# B&R Automation Studio project Soiled_PLC (part 12)

#### ClientPanel.ab - Implementation code
```automation-basic
(********************************************************************
 * COPYRIGHT --
 ********************************************************************
 * Program: ClientPanel
 * File: ClientPanel.ab
 * Author: Dave
 * Created: December 09, 2010
 ********************************************************************
 * Implementation of program ClientPanel
 ********************************************************************)

;Version 1.00 12/12/2010 D.J. First Issue

PROGRAM _INIT

	ColdStart	= FALSE
	panelStatus = 0

	;Set IF port number for panel
	strcpy(ADR(ClientGeneral.IFport),"IF1")

END_PROGRAM

PROGRAM _CYCLIC

	;Read system information

	IF (panelStatus = 0) THEN

		IF (ClientGeneral.ChangePage <> 0) THEN
			ClientGeneral.ChangePage 	= 0 ;Set Init_Page
			ClientGeneral.ButtonPressed = 0 ;Clear button pressed
		ENDIF

		panelStatus = panelStatus + 1

	ENDIF

	;Read IP Address
	IF (panelStatus = 1) THEN

		CfgGetIPAddr_0.enable 	= TRUE
		CfgGetIPAddr_0.pDevice 	= ADR(ClientGeneral.IFport)
		CfgGetIPAddr_0.pIPAddr 	= ADR(ClientGeneral.IPaddress)
		CfgGetIPAddr_0.Len 		= SIZEOF(ClientGeneral.IPaddress)
		CfgGetIPAddr_0 FUB CfgGetIPAddr()

		IF CfgGetIPAddr_0.status = 0 THEN
			panelStatus = panelStatus + 1
		ELSE IF CfgGetIPAddr_0.status = cfgERR_DEVICE_NOT_EXIST THEN
			strcpy(ADR(ClientGeneral.IFport),"IF5") ;Try different port address IF1 = PCT03 and IF5 = CTT11
		ENDIF

	ENDIF

	;Read Subnet Mask
	IF (panelStatus = 2) THEN

		CfgGetSubnetMask_0.enable 		= TRUE
		CfgGetSubnetMask_0.pDevice 		= ADR(ClientGeneral.IFport)
		CfgGetSubnetMask_0.pSubnetMask 	= ADR(ClientGeneral.SubnetMask)
		CfgGetSubnetMask_0.Len 			= SIZEOF(ClientGeneral.SubnetMask)
		CfgGetSubnetMask_0 FUB CfgGetSubnetMask()

		IF CfgGetSubnetMask_0.status = 0 THEN
			panelStatus = panelStatus + 1
		ENDIF

	ENDIF

	;Read Gateway
	IF (panelStatus = 3) THEN

		CfgGetDefaultGateway_0.enable 	= TRUE
		CfgGetDefaultGateway_0.pDevice 	= ADR(ClientGeneral.IFport)
		CfgGetDefaultGateway_0.pGateway = ADR(ClientGeneral.Gateway)
		CfgGetDefaultGateway_0.Len 		= SIZEOF(ClientGeneral.Gateway)
		CfgGetDefaultGateway_0 FUB CfgGetDefaultGateway()

		IF CfgGetDefaultGateway_0.status = 0 THEN
			panelStatus = panelStatus + 1
		ENDIF

	ENDIF

	;Read Broadcast address
	IF (panelStatus = 4) THEN

		CfgGetBroadcastAddr_0.enable 			= TRUE
		CfgGetBroadcastAddr_0.pDevice 			= ADR(ClientGeneral.IFport)
		CfgGetBroadcastAddr_0.pBroadcastAddr 	= ADR(ClientGeneral.BroadcastAddress)
		CfgGetBroadcastAddr_0.Len 				= SIZEOF(ClientGeneral.BroadcastAddress)
		CfgGetBroadcastAddr_0 FUB CfgGetBroadcastAddr()

		IF CfgGetBroadcastAddr_0.status = 0 THEN
			panelStatus = panelStatus + 1
			ClientGeneral.ChangePage 	= 1	;Set Config Button Page
		ENDIF

	ENDIF

	;Init_Page Time Out
	TON_10ms_0.IN = (panelStatus = 5)
	TON_10ms_0.PT = 1000
	TON_10ms_0 FUB TON_10ms()

	TimedOut = TON_10ms_0.Q

	IF (panelStatus = 5) OR (panelStatus = 20) THEN
		IF (ClientGeneral.ButtonPressed = 1) THEN
			panelStatus 				= 6
			ClientGeneral.ChangePage 	= 2	;Set Password page
			ClientGeneral.ButtonPressed = 0
		ELSE IF TimedOut THEN
			panelStatus 				= 20
		ENDIF
	ENDIF

	;Password Page
	IF (panelStatus = 6)   THEN
		IF (ClientGeneral.ButtonPressed = 2) THEN
			panelStatus 				= 5
			ClientGeneral.ChangePage 	= 1	;Set Config Button Page
			ClientGeneral.ButtonPressed = 0
		ENDIF
		IF ClientGeneral.Password = 7701 THEN
			ClientGeneral.ChangePage 	= 3	;Config Page
			panelStatus 				= 7
		ENDIF
	ENDIF

	;Config Page
	IF (panelStatus = 7) THEN
		IF (ClientGeneral.ButtonPressed = 3)  THEN
			panelStatus 				= 11
			ClientGeneral.ButtonPressed = 0
		ENDIF
	ENDIF

	;Store configuration
	;-------------------

	;Store IP Address
	IF (panelStatus = 11) THEN

		CfgSetIPAddr_0.enable 	= TRUE
		CfgSetIPAddr_0.pDevice 	= ADR(ClientGeneral.IFport)
		CfgSetIPAddr_0.pIPAddr 	= ADR(ClientGeneral.IPaddress)
		CfgSetIPAddr_0.Option 	= cfgOPTION_NON_VOLATILE
		CfgSetIPAddr_0 FUB CfgSetIPAddr()

		IF CfgSetIPAddr_0.status = 0 THEN
			panelStatus = 12
		ELSE IF CfgSetIPAddr_0.status = ERR_FUB_BUSY THEN
			; Busy do Nothing
		ELSE IF CfgSetIPAddr_0.status <> ERR_FUB_BUSY THEN
			panelStatus = 12  	;Ignore Errors
		ENDIF

	ENDIF

	;Write Subnet Mask
	IF (panelStatus = 12) THEN

		CfgSetSubnetMask_0.enable 		= TRUE
		CfgSetSubnetMask_0.pDevice 		= ADR(ClientGeneral.IFport)
		CfgSetSubnetMask_0.pSubnetMask 	= ADR(ClientGeneral.SubnetMask)
		CfgSetSubnetMask_0.Option 		= cfgOPTION_NON_VOLATILE
		CfgSetSubnetMask_0 FUB CfgSetSubnetMask()

		IF CfgSetSubnetMask_0.status = 0 THEN
			panelStatus = 13
		ELSE IF CfgSetSubnetMask_0.status = ERR_FUB_BUSY THEN
			; Busy do Nothing
		ELSE IF CfgSetSubnetMask_0.status <> ERR_FUB_BUSY THEN
			panelStatus = 13 	;Ignore Errors
		ENDIF

	ENDIF

	;Write Gateway
	IF (panelStatus = 13) THEN

		CfgSetDefaultGateway_0.enable 	= TRUE
		CfgSetDefaultGateway_0.pDevice 	= ADR(ClientGeneral.IFport)
		CfgSetDefaultGateway_0.pGateway = ADR(ClientGeneral.Gateway)
		CfgSetDefaultGateway_0.Option 	= cfgOPTION_NON_VOLATILE
		CfgSetDefaultGateway_0 FUB CfgSetDefaultGateway()

		IF CfgSetDefaultGateway_0.status = 0 THEN
			panelStatus = 14
		ELSE IF CfgSetDefaultGateway_0.status = ERR_FUB_BUSY THEN
			; Busy do Nothing
		ELSE IF CfgSetDefaultGateway_0.status <> ERR_FUB_BUSY THEN
			panelStatus = 14	 ;Ignore Errors
		ENDIF

	ENDIF

	;Write Broadcast address
	IF (panelStatus = 14) THEN

		CfgSetBroadcastAddr_0.enable 			= TRUE
		CfgSetBroadcastAddr_0.pDevice 			= ADR(ClientGeneral.IFport)
		CfgSetBroadcastAddr_0.pBroadcastAddr 	= ADR(ClientGeneral.BroadcastAddress)
		CfgSetBroadcastAddr_0.Option 			= cfgOPTION_NON_VOLATILE
		CfgSetBroadcastAddr_0 FUB CfgSetBroadcastAddr()

		IF CfgSetBroadcastAddr_0.status = 0 THEN
			IF ColdStart THEN
				SysResetStatus = SYSreset(TRUE,2) ;Cold Start after changing IP address
			ELSE
				panelStatus = 20
			ENDIF
		ELSE IF CfgSetBroadcastAddr_0.status = ERR_FUB_BUSY THEN
			; Busy do Nothing
		ELSE IF CfgSetBroadcastAddr_0.status <> ERR_FUB_BUSY THEN
			IF ColdStart THEN
				SysResetStatus = SYSreset(TRUE,2) ;Cold Start after changing IP address
			ELSE
				panelStatus = 20 ;Ignore Errors
			ENDIF
		ENDIF

	ENDIF

	;Main Display Page
	IF (panelStatus = 20) THEN
		IF ClientReceive[0].MainDisplay = 0 THEN
			IF ((ClientGeneral.ChangePage <> 20) AND (ClientGeneral.CurrentPage <> 20) AND (ClientGeneral.CurrentPage <> 5)) THEN
				ClientGeneral.ChangePage = 20	;Set Default Main display page
			ENDIF
		ELSE IF ClientReceive[0].MainDisplay > 20 THEN
			IF ((ClientGeneral.ChangePage <> ClientReceive[0].MainDisplay) AND (ClientGeneral.CurrentPage <> ClientReceive[0].MainDisplay)) THEN
				ClientGeneral.ChangePage = ClientReceive[0].MainDisplay	;Set Main display page
			ENDIF
		ENDIF

		;Brightness Adjustment required?
		myBrightness = UDINT(ClientReceive[0].Brightness)
		IF (pnlBrightness <> myBrightness) THEN
			panelStatus = 21
		ENDIF

		;New IP address received
		length = strlen(ADR(ClientReceive[0].IP_Address))
		IF (length > 0) THEN
			;Copy new address before ClientReceive[0].IP_Address is cleared by the server
			strcpy(ADR(NewIPAddress),ADR(ClientReceive[0].IP_Address))
			;New IP Address is the actual Gateway
			strcpy(ADR(ClientGeneral.Gateway),ADR(ClientReceive[0].IP_Address))
			panelStatus = 31 ;Change IP Address
		ENDIF

	ENDIF

	;Remote cold Start
	IF (ClientReceive[0].SYSreset > 0) THEN
		SysResetStatus = SYSreset(TRUE,2) ;Cold Start
	ENDIF

	;Display Brightness
	IF (panelStatus = 21) THEN

		IF myVC_Handle = 0 THEN
			myVC_Handle = VA_Setup(TRUE, "Data1")
		ENDIF
		IF (myVC_Handle > 0) THEN
			IF VA_Saccess(TRUE,myVC_Handle) = 0 THEN
				VA_SetBrightness(TRUE,myVC_Handle,myBrightness)
				VA_SetBacklight(TRUE,myVC_Handle,(myBrightness > 0))
				pnlBrightness = myBrightness
				VA_Srelease(TRUE,myVC_Handle)
			ENDIF
		ENDIF

		panelStatus = 20
	ELSE
		myVC_Handle = 0
	ENDIF

	;Change IP Address
	IF (panelStatus = 31) THEN

		IP_Replace_0.pIP_New = ADR(NewIPAddress)
		IP_Replace_0.pIP_Now = ADR(ClientGeneral.IPaddress)
		IP_Replace_0 FUB IP_Replace()

		IF IP_Replace_0.status = 0 THEN
			ClientGeneral.IPaddress = IP_Replace_0.IP_Replace
			panelStatus = 32
		ELSE
			panelStatus = 20
		ENDIF

	ENDIF

	;Change Gateway
	IF (panelStatus = 32) THEN

		;IP_Replace_0.pIP_New = ADR(NewIPAddress)
		;IP_Replace_0.pIP_Now = ADR(ClientGeneral.Gateway)
		;IP_Replace_0 FUB IP_Replace()

		;IF IP_Replace_0.status = 0 THEN
		;	ClientGeneral.Gateway = IP_Replace_0.IP_Replace
			panelStatus = 33
		;ELSE
		;	panelStatus = 20
		;ENDIF

	ENDIF

	;Change Broadcast Address
	IF (panelStatus = 33) THEN

		IP_Replace_0.pIP_New = ADR(NewIPAddress)
		IP_Replace_0.pIP_Now = ADR(ClientGeneral.BroadcastAddress)
		IP_Replace_0 FUB IP_Replace()

		IF IP_Replace_0.status = 0 THEN
			ClientGeneral.BroadcastAddress = IP_Replace_0.IP_Replace
			panelStatus = 34
		ELSE
			panelStatus = 20
		ENDIF

	ENDIF

	;Change Server IP
	IF (panelStatus = 34) THEN

		IP_Replace_0.pIP_New = ADR(NewIPAddress)
		IP_Replace_0.pIP_Now = ADR(ClientServerIP)
		IP_Replace_0 FUB IP_Replace()

		IF IP_Replace_0.status = 0 THEN
			ClientServerIP 	= IP_Replace_0.IP_Replace
			ColdStart		= TRUE
			panelStatus 	= 11 ;Store New Values
		ELSE
			panelStatus = 20
		ENDIF

	ENDIF

END_PROGRAM
```

#### ClientPanel.var - Local variables
```iecst
(********************************************************************
 * COPYRIGHT --
 ********************************************************************
 * Program: ClientPanel
 * File: ClientPanel.var
 * Author: Dave
 * Created: December 09, 2010
 ********************************************************************
 * Local variables of program ClientPanel
 ********************************************************************)
VAR
	panelStatus : UINT;
	CfgGetIPAddr_0 : CfgGetIPAddr;
	CfgGetSubnetMask_0 : CfgGetSubnetMask;
	CfgGetDefaultGateway_0 : CfgGetDefaultGateway;
	CfgGetBroadcastAddr_0 : CfgGetBroadcastAddr;
	TON_10ms_0 : TON_10ms;
	TimedOut : BOOL;
	CfgSetIPAddr_0 : CfgSetIPAddr;
	CfgSetSubnetMask_0 : CfgSetSubnetMask;
	CfgSetDefaultGateway_0 : CfgSetDefaultGateway;
	CfgSetBroadcastAddr_0 : CfgSetBroadcastAddr;
	SysResetStatus : UINT;
	myVC_Handle : UDINT;
	myBrightness : UDINT;
	pnlBrightness : UDINT;
	length : UINT;
	IP_Replace_0 : IP_Replace;
	ColdStart : BOOL;
	NewIPAddress : STRING[16];
END_VAR
```

### Program Logical/Displays/Client (IEC, version 1.00.0) - AsTCP Diplay Client

#### Client.ab - Implementation code
```automation-basic
(********************************************************************
 * COPYRIGHT --
 ********************************************************************
 * Program: Client
 * File: Client.ab
 * Author: Dave
 * Created: December 06, 2010
 ********************************************************************
 * Implementation of program Client
 ********************************************************************)

;Version 1.00 12/12/2010 D.J. First Issue
;Version 2.00 22/07/2011 D.J. Added sckWaitSync - Improve Sync between Slave and Master

PROGRAM _INIT

	IF ((IdentRetain > 0) AND (Client.TcpOpen_0.ident = 0)) THEN
		Client.TcpOpen_0.ident = IdentRetain
	ENDIF

END_PROGRAM

PROGRAM _CYCLIC
	ClientText
	;Sending and Recieving Syc / Speed from Server
	ScanClock 		= clock_ms()
	ScanNow 		= (ScanClock - ScanLastClock)
	ScanLastClock 	= ScanClock
	ScanCount 		= (ScanCount + UINT(ScanNow))

	;Init Ethernet Socket - Pause after any close etc
	TON_10ms_0.IN = (SocketState = sckClosed)
	TON_10ms_0.PT = 100
	TON_10ms_0 FUB TON_10ms()

	IF TON_10ms_0.Q THEN
		SocketState = sckConnecting
	ENDIF

	;Close Ethernet Socket
	IF SocketState = sckError THEN

		Client.TcpClose_0.enable 	= TRUE
		Client.TcpClose_0.ident 	= Client.TcpOpen_0.ident
		Client.TcpClose_0.how 		= 0						;tcpSHUT_RD OR tcpSHUT_WR;
		Client.TcpClose_0 FUB TcpClose()

		IF Client.TcpClose_0.status = 0 THEN
			SocketState = sckClosed
		ELSE IF Client.TcpClose_0.status = ERR_FUB_BUSY THEN
		 	;Busy
		ELSE IF Client.TcpClose_0.status = tcpERR_INVALID_IDENT THEN
			SocketState = sckClosed
		ELSE IF Client.TcpClose_0.status = tcpERR_NOT_CONNECTED THEN
			SocketState = sckClosed
		ELSE IF Client.TcpOpen_0.status <> ERR_FUB_BUSY THEN
			SocketState = sckConnecting
		ENDIF

	ENDIF

	;Open Ethernet Socket
	IF SocketState = sckConnecting THEN
		Client.TcpOpen_0.enable  	= TRUE
		Client.TcpOpen_0.pIfAddr 	= 0					;Which Interface to open
		Client.TcpOpen_0.port 		= 12001				;Client Port
		Client.TcpOpen_0.options 	= 0
		Client.TcpOpen_0 FUB TcpOpen()

		IF Client.TcpOpen_0.status = 0 THEN
			SocketState = sckSetLinger ;sckConnected
			IdentRetain = Client.TcpOpen_0.ident
		ELSE IF Client.TcpOpen_0.status = ERR_FUB_BUSY THEN
		 	;Busy
		ELSE IF Client.TcpOpen_0.status = tcpERR_ALREADY_EXIST THEN
			SocketState = sckError
		ELSE IF Client.TcpOpen_0.status = tcpERR_SOCKET_BIND THEN
			SocketState = sckError
		ELSE
			SocketState = sckError
		ENDIF
	ENDIF

	;Set Open Linger Options
	IF SocketState = sckSetLinger THEN

		Client.linger_opt.lLinger 	= 0 ;Linger Time = 0
		Client.linger_opt.lOnOff	= 1	;Linger Option On

		Client.TcpIoctl_0.enable 	= TRUE
		Client.TcpIoctl_0.ident 	= Client.TcpOpen_0.ident
		Client.TcpIoctl_0.ioctl		= tcpSO_LINGER_SET
		Client.TcpIoctl_0.pData		= ADR(Client.linger_opt)
		Client.TcpIoctl_0.datalen 	= SIZEOF(Client.linger_opt)
		Client.TcpIoctl_0 FUB TcpIoctl()

		IF Client.TcpIoctl_0.status = 0 THEN
			SocketState = sckConnected
		ELSE IF Client.TcpIoctl_0.status = ERR_FUB_BUSY THEN  (* TcpIoctl not finished -> redo *)
			;Busy
		ELSE
			SocketState = sckError
		ENDIF
	ENDIF

	;Connect to server
	IF SocketState = sckConnected THEN

		Client.TcpClient_0.enable 	= TRUE
		Client.TcpClient_0.ident 	= Client.TcpOpen_0.ident 	;Connection Ident from AsTCP.TCP_Open
		Client.TcpClient_0.portserv = 12000						;Server port number
		Client.TcpClient_0.pServer 	= ADR(ClientServerIP)			;Server IP Adderss
		Client.TcpClient_0 FUB TcpClient()

		IF Client.TcpClient_0.status = 0 THEN
			SocketState = sckSend
		ELSE IF Client.TcpClient_0.status = ERR_FUB_BUSY THEN
			;Busy
		ELSE IF Client.TcpClient_0.status = tcpERR_INVALID THEN
			SocketState = sckError
		ELSE IF Client.TcpClient_0.status = tcpERR_NOT_CONNECTED THEN
			SocketState = sckClosed
		ELSE
			SocketState = sckError
		ENDIF

	ENDIF

	;Send Data
	IF SocketState = sckSend THEN

		Client.TcpSend_0.enable 	= TRUE
		Client.TcpSend_0.ident 		= Client.TcpOpen_0.ident
		Client.TcpSend_0.pData 		= ADR(ClientSend)	;Address of send data
		Client.TcpSend_0.datalen 	= SIZEOF(ClientSend);Length of send data
		Client.TcpSend_0.flags 		= 0
		Client.TcpSend_0 FUB TcpSend()

		IF Client.TcpSend_0.status = 0 THEN
			SocketState = sckReceive
		ELSE IF Client.TcpSend_0.status = ERR_FUB_BUSY THEN
			;Busy
		ELSE IF (Client.TcpSend_0.status = tcpERR_SENTLEN) OR (Client.TcpSend_0.status = tcpERR_NOT_CONNECTED) THEN
			SocketState = sckError
		ELSE
			SocketState = sckError
		ENDIF

	ENDIF

	IF SocketState = sckReceive THEN

		Client.TcpRecv_0.enable 	= TRUE
		Client.TcpRecv_0.ident 		= Client.TcpOpen_0.ident			;Connection Ident from AsTCP.TCP_Open
		Client.TcpRecv_0.pData		= ADR(ClientReceive)	;Where to store the incoming data
		Client.TcpRecv_0.datamax 	= SIZEOF(ClientReceive)	;Lenght of data buffer
		Client.TcpRecv_0.flags 		= 0
		Client.TcpRecv_0 FUB TcpRecv()

		IF Client.TcpRecv_0.status = 0 THEN  (* Data was received sucessfully -> Send next packet *)
			SocketState 			= sckWaitSync
		ELSE IF Client.TcpRecv_0.status = tcpERR_NO_DATA THEN  (* No data received - wait *)
		    IF Client.recv_timeout > 10 THEN
 		    	SocketState = sckError
		  	ENDIF
		ELSE IF Client.TcpRecv_0.status = ERR_FUB_BUSY THEN
			;Busy
		ELSE IF Client.TcpRecv_0.status = tcpERR_NOT_CONNECTED THEN
			SocketState = sckError
		ELSE
			SocketState = sckError
		ENDIF

		Client.recv_timeout = Client.recv_timeout + 1
	ELSE IF SocketState <> sckReceive THEN
		Client.recv_timeout = 0
	ENDIF

	;Wait until SyncStart (Master controls the connection communication speed)
	IF SocketState = sckWaitSync THEN
		IF (ScanCount >= ClientReceive[0].CycleSync_ms) THEN
			ScanCount 	= 0
			SocketState	= sckSend
		ENDIF
	ENDIF

END_PROGRAM
```

#### Client.typ - Local data types
```iecst
(********************************************************************
 * COPYRIGHT --
 ********************************************************************
 * Program: Client
 * File: Client.typ
 * Author: Dave
 * Created: December 06, 2010
 ********************************************************************
 * Local data types of program Client
 ********************************************************************)

TYPE
	Client_typ : 	STRUCT  (*TCP Client Variables*)
		TcpOpen_0 : TcpOpen; (*AsTCP.TcpOpen FUB*)
		TcpClient_0 : TcpClient; (*AsTCP.TcpClient FUB*)
		TcpRecv_0 : TcpRecv; (*AsTCP.TcpRecv FUB*)
		TcpSend_0 : TcpSend; (*AsTCP.TcpSend FUB*)
		TcpIoctl_0 : TcpIoctl; (*AsTCP.TcpIoctl FUB*)
		TcpClose_0 : TcpClose; (*AsTCP.TcpClose FUB*)
		linger_opt : tcpLINGER_typ; (*AsTCP.tcpLINGER_typ*)
		recv_timeout : UDINT; (*receive timeout*)
	END_STRUCT;
END_TYPE
```

#### Client.var - Local variables
```iecst
(********************************************************************
 * COPYRIGHT --
 ********************************************************************
 * Program: Client
 * File: Client.var
 * Author: Dave
 * Created: December 06, 2010
 ********************************************************************
 * Local variables of program Client
 ********************************************************************)
VAR
	ScanCount : UINT;
	ScanClock : TIME;
	ScanLastClock : TIME;
	ScanNow : TIME := T#0ms;
	Client : Client_typ;
END_VAR
VAR RETAIN
	IdentRetain : UDINT;
END_VAR
VAR
	SocketState : USINT;
END_VAR
VAR CONSTANT
	sckClosed : USINT := 0;
	sckConnecting : USINT := 1;
	sckConnected : USINT := 2;
	sckError : USINT := 3;
	sckListening : USINT := 4;
	sckReceive : USINT := 5;
	sckSend : USINT := 6;
	sckSetLinger : USINT := 7;
	sckWaitSync : USINT := 8;
END_VAR
VAR
	TON_10ms_0 : TON_10ms;
	ReadWriteEnable : BOOL;
	SyncStart : BOOL;
END_VAR
```

### Program Logical/Displays/ClientDataEntry (IEC) - Client Panel Data Entry

#### ClientDataEntry.ab - Cyclic code
```automation-basic
(********************************************************************
 * COPYRIGHT --
 ********************************************************************
 * Program: ClientDataEntry
 * File: ClientDataEntry.ab
 * Author: Dave
 * Created: October 17, 2011
 ********************************************************************
 * Implementation of program ClientDataEntry
 ********************************************************************)

PROGRAM _CYCLIC

	IF (ClientDataLocal[0].Start > 0) THEN
		ClientSend[0].Command = 1 ;Start Button Pressed
	;ELSE IF (ClientDataLocal[0].Start > 0) THEN
	;	ClientSend[0].Command = 2 ;Add more buttons if required
	ELSE
		ClientSend[0].Command = 0
	ENDIF

END_PROGRAM
```

#### ClientDataEntry.typ - Local data types
```iecst
(********************************************************************
 * COPYRIGHT --
 ********************************************************************
 * Program: ClientDataEntry
 * File: ClientDataEntry.typ
 * Author: Dave
 * Created: October 17, 2011
 ********************************************************************
 * Local data types of program ClientDataEntry
 ********************************************************************)

TYPE
	ClientDataEntry_typ : 	STRUCT
		Start : UINT;
	END_STRUCT;
END_TYPE
```

#### ClientDataEntry.var - Local variables
```iecst
(********************************************************************
 * COPYRIGHT --
 ********************************************************************
 * Program: ClientDataEntry
 * File: ClientDataEntry.var
 * Author: Dave
 * Created: October 17, 2011
 ********************************************************************
 * Local variables of program ClientDataEntry
 ********************************************************************)
VAR
	ClientDataLocal : ARRAY[0..3] OF ClientDataEntry_typ;
	n : UINT;
END_VAR
```

### Package Logical/Displays/myPanel - General Use Panel

### my_Panel.typ - Global data types
```iecst
(********************************************************************
 * COPYRIGHT --
 ********************************************************************
 * Package: myPanel
 * File: myPanel.typ
 * Author: Administrator
 * Created: February 23, 2009
 ********************************************************************
 * Data types of package myPanel
 ********************************************************************)

TYPE
	Panel_typ : 	STRUCT
		Text : STRING[20];
		Datapoint : DINT;
		Min : DINT;
		Max : DINT;
		Status : UINT;
		Completion : UINT;
		Locking : UINT;
	END_STRUCT;
	Panel_Motor_Monitor_typ : 	STRUCT
		MonitorIndex : USINT;
		Datapoint : DINT;
	END_STRUCT;
END_TYPE
```

### my_Panel.var - Global variables
```iecst
(********************************************************************
 * COPYRIGHT --
 ********************************************************************
 * Package: myPanel
 * File: myPanel.var
 * Author: Administrator
 * Created: February 23, 2009
 ********************************************************************
 * Variables of package myPanel
 ********************************************************************)
VAR
	PanelData : ARRAY[0..20] OF Panel_typ := [21(0)];
END_VAR
```

- Visualisation Logical/Displays/myPanel/myDataEntry1 (not shown)

### Program Logical/Displays/myPanel/myPanel (IEC) - General Use Panel Display

#### myPanel.var - Local variables
```iecst
(********************************************************************
 * COPYRIGHT --
 ********************************************************************
 * Program: myPanel
 * File: myPanel.var
 * Author: Administrator
 * Created: February 23, 2009
 ********************************************************************
 * Local variables of program myPanel
 ********************************************************************)
VAR
	myDINT : DINT;
	myString : ARRAY[0..9] OF USINT;
	Length : UINT;
END_VAR
```

#### myPanelCyclic.ab - Cyclic code
```automation-basic
(********************************************************************
 * COPYRIGHT --
 ********************************************************************
 * Program: myPanel
 * File: myPanelCyclic.ab
 * Author: Administrator
 * Created: February 23, 2009
 ********************************************************************
 * Implementation of program myPanel
 ********************************************************************)

PROGRAM _CYCLIC

	;----------
	;SVC6 Panel
	;----------

	strcpy(ADR(PanelData[1].Text),"Sortierstand")
	;memcpy(ADR(PanelData[1].Text),ADR(zzGetNamesData[2].CatName),20)

	PanelData[1].Min 		= 0
	PanelData[1].Max		= Std.MaxCats
	PanelData[1].Locking 	= 0 ;0 = Locked

	IF (PanelData[1].Completion = 1) THEN
		;D[701] = PanelData[1].Datapoint
		PanelData[1].Completion = 0
	ELSE
		;Show Data Here
		PanelData[1].Datapoint = DINT(Bag[199].Cat)
	ENDIF

	;strcpy(ADR(PanelData[2].Text),"Category")
	memcpy(ADR(PanelData[2].Text),ADR(zzGetNamesData[2].CusName),20)

	PanelData[2].Min 		= 0
	PanelData[2].Max		= Std.MaxCust
	PanelData[2].Locking 	= 0 ; 0 = Locked

	IF (PanelData[2].Completion = 1) THEN
		;Bag[399].Cat = UDINT(PanelData[2].Datapoint)
		PanelData[2].Completion = 0
	ELSE
		;Show Data Here
		PanelData[2].Datapoint = DINT(Bag[199].Cus)
	ENDIF

	strcpy(ADR(PanelData[3].Text),"Beladeband")
	;memcpy(ADR(PanelData[3].Text),ADR(zzGetNamesData[1].CatName),20)

	PanelData[3].Min 		= 0
	PanelData[3].Max		= Std.MaxCats
	PanelData[3].Locking 	= 1 ; 0 = Locked

	IF (PanelData[3].Completion = 1) THEN

		Bag[198].Cat = UDINT(PanelData[3].Datapoint)
		PanelData[3].Completion = 0
	ELSE
		;Show Data Here
		Bag[198].Prg = USINT(zzGetDBData[2].Prg)
		PanelData[3].Datapoint = DINT(Bag[198].Cat)
	ENDIF

	;strcpy(ADR(PanelData[4].Text),"Destination")

	memcpy(ADR(PanelData[4].Text),ADR(zzGetNamesData[1].CusName),20)

	PanelData[4].Min 		= 0
	PanelData[4].Max		= Std.MaxCust
	PanelData[4].Locking 	= NOT (SB2Status = 2);1 ; 0 = Locked

	IF (PanelData[4].Completion = 1) THEN
		Bag[198].Cus = UDINT(PanelData[4].Datapoint)
		PanelData[4].Completion = 0
	ELSE
		;Show Data Here
		PanelData[4].Datapoint = DINT(Bag[198].Cus)
	ENDIF

	;Weight
	;Length = itoa(DINT(Bag[399].Wgt / 10),ADR(myString))
	;strcpy(ADR(myString[Length]),"kg")

	;strcpy(ADR(PanelData[5].Text),ADR(myString))
	strcpy(ADR(PanelData[5].Text),"Beladeband")

	IF EDGEPOS(PanelData[5].Status = 1) AND (D[11] = 0) THEN
		D[11] = TRUE
	ELSE IF EDGEPOS(PanelData[5].Status = 0) AND (D[11] = 1) THEN
		D[11] = FALSE
	ENDIF
			PanelData[5].Status = D[11]
	;Messages
	IF SB2Status = 0 THEN
		strcpy(ADR(PanelData[6].Text),"Bereit")
	ELSE IF SB2Status = 1 THEN
		strcpy(ADR(PanelData[6].Text),"Kundenwechsel -Stopp")
	ELSE IF SB2Status = 2 THEN
		strcpy(ADR(PanelData[6].Text),"Kundenwechsel")
	ELSE IF SB2Status = 7 THEN
		strcpy(ADR(PanelData[6].Text),"Datei nicht gefunden!")
	ENDIF
(*	;Messages
	IF VCStatus[6] = 0 THEN
		strcpy(ADR(PanelData[6].Text),"")
	ELSE IF VCStatus[6] = 1 THEN
		strcpy(ADR(PanelData[6].Text),"Destination not valid!")
	ELSE IF VCStatus[6] = 2 THEN
		strcpy(ADR(PanelData[6].Text),"Category not valid!")
	ELSE IF VCStatus[6] = 3 THEN
		strcpy(ADR(PanelData[6].Text),"Customer not valid!")
	ELSE IF VCStatus[6] = 5 THEN
		strcpy(ADR(PanelData[6].Text),"No bag on carriage!")
	ELSE IF VCStatus[6] = 6 THEN
		strcpy(ADR(PanelData[6].Text),"Destination not valid!")
	ELSE IF VCStatus[6] = 7 THEN
		strcpy(ADR(PanelData[6].Text),"Program not valid!")
	ENDIF
*)
	;----------
	;SLU1 Panel
	;----------

	strcpy(ADR(PanelData[11].Text),"Program")

	PanelData[11].Min 		= 0
	PanelData[11].Max		= 99
	PanelData[11].Locking 	= 0 ;0 = Locked

	IF (PanelData[11].Completion = 1) THEN
		;D[701] = PanelData[1].Datapoint
		PanelData[11].Completion = 0
	ELSE
		;Show Data Here
		PanelData[11].Datapoint = DINT(Bag[400].Prg)
	ENDIF

	strcpy(ADR(PanelData[12].Text),"Category")

	PanelData[12].Min 		= 0
	PanelData[12].Max		= Std.MaxCats
	PanelData[12].Locking 	= 1 ; 0 = Locked

	IF (PanelData[12].Completion = 1) THEN
		Bag[400].Cat = UDINT(PanelData[12].Datapoint)
		PanelData[12].Completion = 0
	ELSE
		;Show Data Here
		PanelData[12].Datapoint = DINT(Bag[400].Cat)
	ENDIF

	strcpy(ADR(PanelData[13].Text),"Customer")

	PanelData[13].Min 		= 0
	PanelData[13].Max		= Std.MaxCust
	PanelData[13].Locking 	= 1 ; 0 = Locked

	IF (PanelData[13].Completion = 1) THEN
		Bag[400].Cus = UDINT(PanelData[13].Datapoint)
		PanelData[13].Completion = 0
	ELSE
		;Show Data Here
		PanelData[13].Datapoint = DINT(Bag[400].Cus)
	ENDIF

	strcpy(ADR(PanelData[14].Text),"Destination")

	PanelData[14].Min 		= 0
	PanelData[14].Max		= 99
	PanelData[14].Locking 	= 1 ; 0 = Locked

	IF (PanelData[14].Completion = 1) THEN
		Bag[400].Dst = USINT(PanelData[14].Datapoint)
		PanelData[14].Completion = 0
	ELSE
		;Show Data Here
		PanelData[14].Datapoint = DINT(Bag[400].Dst)
	ENDIF

		;Weight
	Length = itoa(DINT(Bag[400].Wgt / 10),ADR(myString))
	strcpy(ADR(myString[Length]),"kg")

	strcpy(ADR(PanelData[15].Text),ADR(myString))

	;Messages
	IF SB2Status = 0 THEN
		strcpy(ADR(PanelData[16].Text),"")
	ELSE IF SB2Status = 1 THEN
		strcpy(ADR(PanelData[16].Text),"Linen Over-Weight")
	ELSE IF SB2Status = 7 THEN
		strcpy(ADR(PanelData[16].Text),"Program not valid!")
	ENDIF

END_PROGRAM
```

- Changing Display Size PCT03 and CTT11.doc (binary file, 20992 bytes)
### Library Logical/Displays/DispLib (IEC) - Displays Functions Library

#### DispLib.fun - Exported functions and function blocks
```iecst
(********************************************************************
 * COPYRIGHT --
 ********************************************************************
 * Library: DispLib
 * File: DispLib.fun
 * Author: Dave
 * Created: December 12, 2010
 ********************************************************************
 * Functions and function blocks of library DispLib
 ********************************************************************)

FUNCTION_BLOCK IP_Replace (*Replace existing first 3 parts of IP address*)
	VAR_INPUT
		pIP_New : UDINT;
		pIP_Now : UDINT;
	END_VAR
	VAR_OUTPUT
		IP_Replace : STRING[16];
		status : UINT;
	END_VAR
	VAR
		ethStatus : UINT;
		Node : UDINT;
		IP_Hex : UDINT;
		IP_Build : UDINT;
		IP_HexReplace : UDINT;
		IP_HexNew : UDINT;
	END_VAR
END_FUNCTION_BLOCK
```

#### IP_Replace.ab - Replace existing first 3 parts of IP address
```automation-basic
(********************************************************************
 * COPYRIGHT --
 ********************************************************************
 * Library: DispLib
 * File: IP_Replace.ab
 * Author: Dave
 * Created: December 12, 2010
 ********************************************************************
 * Implementation of library DispLib
 ********************************************************************)

(* Replace existing first 3 parts of IP address *)

;Version 1.00 12/12/2010 D.J. First Issue

FUNCTION_BLOCK IP_Replace

	;Get the node part of the existing IP arddress
	ethStatus 	= ethInetAton(pIP_Now,ADR(IP_Hex))
	Node 		= 0
	IF ethStatus = 0 THEN
		;Get the node number from the IP address
		Node 		= (IP_Hex AND $FF000000) ;Mask out the IP address
	ELSE
		status = 1
	ENDIF

	;Get the new IP address first three parts
	IF (Node > 0) THEN
		ethStatus 	= ethInetAton(pIP_New,ADR(IP_HexNew))
		IP_Build 	= 0
		IF ethStatus = 0 THEN
			;Get the node number from the IP address
			IP_Build	= (IP_HexNew AND $00FFFFFF) ;Mask out the node part of the address
		ELSE
			status = 3
		ENDIF
	ELSE
		status = 2
	ENDIF

	;Build the complete replacement IP address
	IF ((Node > 0) AND (IP_Build > 0)) THEN
		IP_HexReplace 	= (IP_Build + Node)
		ethStatus = ethInetNtoa(IP_HexReplace,ADR(IP_Replace))
		IF ethStatus = 0 THEN
			status = 0
		ENDIF
	ELSE
		status = 4
	ENDIF

END_FUNCTION_BLOCK
```

### Data object Logical/Displays/svc1 (Vc3) - Visualization

- SVC3.bak (binary file, 197042 bytes)
- Program Logical/SQL/SQLReadWriteTest (IEC) (no source held here)

- Program Logical/SQL/Test_bagMaint (IEC) (no source held here)

### Program Logical/SQL/zzGetNamesSQL/zzGetNameSQL (IEC) - Get Names for Display

#### zzGetNames.var - Local variables
```iecst
(********************************************************************
 * COPYRIGHT --
 ********************************************************************
 * Program: zzGetNames
 * File: zzGetNames.var
 * Author: Dave
 * Created: November 19, 2010
 ********************************************************************
 * Local variables of program zzGetNames
 ********************************************************************)
VAR
	MaxDisplays : UINT := 4;
	OwnerID : UDINT;
	TviewReplyOwnerID : UDINT;
	WaitReply : BOOL;
	myBag : UINT;
	CommsID : UDINT;
	Timer2Q : BOOL;
	Timer1Q : BOOL;
	Timer1ET : UDINT;
	Timer2ET : UDINT;
	result : DINT;
	TestTim : UDINT;
	mySql : UINT;
	myPrgString : STRING[24];
	myCatString : STRING[24];
	myCusString : STRING[24];
	SqlWriteActive : BOOL;
	RefreshDataTest : BOOL;
	n : INT;
END_VAR
```

#### zzGetNames.ab - Implementation code
```automation-basic
(********************************************************************
 * COPYRIGHT --
 ********************************************************************
 * Program: zzGetNames
 * File: zzGetNames.ab
 * Author: Dave
 * Created: November 19, 2010
 ********************************************************************
 * Implementation of program zzGetNames
 ********************************************************************)

;Get names from TrackView - Program, Category and Customer

;Version 1.00 19/11/2010 D.J. First Issue
;Version 2.00 12/12/2010 D.J. Added default values
;Version 3.00 19/10/2011 D.J. Clear Name when number has changed - if no TrackView then name will remain clear.

;Enter the required bag numbers for collection of names. Use the resulting names in transmisions to displays.

PROGRAM _INIT
	mySql = 96
	MaxDisplays = 1
	LOOP n = 1 TO MaxDisplays DO
		zzGetNamesData[n].BagNumber = 100 + n
	ENDLOOP
	;zzGetNamesData[20].BagNumber = 194	; Static Bag
	;zzGetNamesData[21].BagNumber = 411	; Customer Change 1
	;zzGetNamesData[22].BagNumber = 412	; Customer Change 2
	;zzGetNamesData[23].BagNumber = 401	; Customer Change Current Cust 1
	;zzGetNamesData[24].BagNumber = 402	; Customer Change Current Cust 2

	IF (MaxDisplays > SIZEOF(zzGetNamesData)) THEN
		MaxDisplays = SIZEOF(zzGetNamesData)
	ENDIF

	WaitReply = FALSE

	zzGetNamesData[0].BagNumber = 1
	zzGetNamesData[0].Prg		= 1
	strcpy(ADR(zzGetNamesData[0].PrgLong),"PRG")
	strcpy(ADR(zzGetNamesData[0].PrgName),"ProgramName")
	zzGetNamesData[0].Cat		= 1
	strcpy(ADR(zzGetNamesData[0].CatLong),"CAT")
	strcpy(ADR(zzGetNamesData[0].CatName),"CategoryName")
	zzGetNamesData[0].Cus		= 1
	strcpy(ADR(zzGetNamesData[0].CusLong),"CUS")
	strcpy(ADR(zzGetNamesData[0].CusName),"CustomerName")

END_PROGRAM

PROGRAM _CYCLIC
	IF RefreshDataTest THEN
		LOOP n = 1 TO MaxDisplays DO
			zzGetNamesData[n].Cat = 0
		ENDLOOP
		RefreshDataTest = FALSE
	ENDIF
	;Clear all display strings while waiting for replies,

	LOOP n = 1 TO MaxDisplays DO
		myBag = zzGetNamesData[n].BagNumber

		IF ((zzGetNamesData[n].Prg <> Bag[myBag].Prg) AND (Bag[myBag].Prg > 0)) THEN
			memcpy(ADR(zzGetNamesData[n].PrgLong),ADR(""),8)
			memcpy(ADR(zzGetNamesData[n].PrgName),ADR(""),32)
		ENDIF

		IF ((zzGetNamesData[n].Cat <> Bag[myBag].Cat) AND (Bag[myBag].Cat > 0)) THEN
			memcpy(ADR(zzGetNamesData[n].CatLong),ADR(""),8)
			memcpy(ADR(zzGetNamesData[n].CatName),ADR(""),32)
		ENDIF

		IF ((zzGetNamesData[n].Cus <> Bag[myBag].Cus) AND (Bag[myBag].Cus > 0)) THEN
			memcpy(ADR(zzGetNamesData[n].CusLong),ADR(""),8)
			memcpy(ADR(zzGetNamesData[n].CusName),ADR(""),32)
		ENDIF
	ENDLOOP

	;Search for display data that needs updating
	IF NOT WaitReply THEN

		OwnerID = OwnerID + 1
		IF (OwnerID > MaxDisplays) THEN
			OwnerID = 1
		ENDIF

		myBag = zzGetNamesData[OwnerID].BagNumber

		IF ((zzGetNamesData[OwnerID].Prg <> Bag[myBag].Prg) AND (Bag[myBag].Prg > 0)) THEN
			memcpy(ADR(zzGetNamesData[OwnerID].PrgLong),ADR(""),8)
			memcpy(ADR(zzGetNamesData[OwnerID].PrgName),ADR(""),32)
			WaitReply = TRUE
		ENDIF

		IF ((zzGetNamesData[OwnerID].Cat <> Bag[myBag].Cat) AND (Bag[myBag].Cat > 0)) THEN
			;Special for Brolli Get Prg code back for Data entry
			IF ((OwnerID = 25) OR (OwnerID = 26)) THEN
				Bag[myBag].Prg = 0
				zzGetNamesData[OwnerID].Prg = 0
				memcpy(ADR(zzGetNamesData[OwnerID].PrgLong),ADR(""),8)
				memcpy(ADR(zzGetNamesData[OwnerID].PrgName),ADR(""),32)
			ENDIF
			memcpy(ADR(zzGetNamesData[OwnerID].CatLong),ADR(""),8)
			memcpy(ADR(zzGetNamesData[OwnerID].CatName),ADR(""),32)
			WaitReply = TRUE
		ELSE IF Bag[myBag].Cat = 0 THEN
			zzGetNamesData[OwnerID].Cat = 0
			strcpy(ADR(zzGetNamesData[OwnerID].CatLong),"")
			strcpy(ADR(zzGetNamesData[OwnerID].CatName),"")
			strcpy(ADR(zzGetNamesData[OwnerID].CusName),"")
			strcpy(ADR(zzGetNamesData[OwnerID].PrgName),"")
			strcpy(ADR(zzGetNamesData[OwnerID].ImagePath),"")
		ENDIF

		IF ((zzGetNamesData[OwnerID].Cus <> Bag[myBag].Cus) AND (Bag[myBag].Cus > 0)) THEN
			memcpy(ADR(zzGetNamesData[OwnerID].CusLong),ADR(""),8)
			memcpy(ADR(zzGetNamesData[OwnerID].CusName),ADR(""),32)
			WaitReply = TRUE
		ENDIF

		;Set TrackView Registers
		IF WaitReply THEN
			itoa(Bag[myBag].Prg,ADR(myPrgString))
			itoa(Bag[myBag].Cat,ADR(myCatString))
			itoa(Bag[myBag].Cus,ADR(myCusString))
			SqlRequest[mySql].Request = TRUE
		ENDIF

	ENDIF

	;Set request to TrackView until reply
	IF (WaitReply AND SqlRequest[mySql].Complete) THEN

		myBag = zzGetNamesData[OwnerID].BagNumber

		strcpy(ADR(zzGetNamesData[OwnerID].PrgLong),ADR(SqlRequest[mySql].OutputData[1]))
		strcpy(ADR(zzGetNamesData[OwnerID].PrgName),ADR(SqlRequest[mySql].OutputData[2]))
		result = strcmp(ADR(zzGetNamesData[OwnerID].PrgName),"ProgCodeReturned")
		IF (result = 0) THEN
			Bag[myBag].Prg = USINT(atoi(ADR(zzGetNamesData[OwnerID].PrgLong)))
		ENDIF
		zzGetNamesData[OwnerID].Prg = Bag[myBag].Prg

		zzGetNamesData[OwnerID].Cat = Bag[myBag].Cat
		strcpy(ADR(zzGetNamesData[OwnerID].CatLong),ADR(SqlRequest[mySql].OutputData[3]))
		strcpy(ADR(zzGetNamesData[OwnerID].CatName),ADR(SqlRequest[mySql].OutputData[4]))

		zzGetNamesData[OwnerID].Cus = Bag[myBag].Cus
		strcpy(ADR(zzGetNamesData[OwnerID].CusLong),ADR(SqlRequest[mySql].OutputData[5]))
		strcpy(ADR(zzGetNamesData[OwnerID].CusName),ADR(SqlRequest[mySql].OutputData[6]))

		strcpy(ADR(zzGetNamesData[OwnerID].ImagePath),ADR(SqlRequest[mySql].OutputData[7]))

		WaitReply 	= FALSE

	ENDIF

IF SqlRequest[mySql].Request AND NOT SqlWriteActive THEN ; Write Count to SQL
	SqlWriteActive = TRUE
	SqlRequest[mySql].SQLType = cSQLType_ReadWrite
	SqlRequest[mySql].SQL_usp = cSQLReq_zzGetNames
	SqlRequest[mySql].NoOfParams = 3

	SqlRequest[mySql].Parameters[0].Type = cSQLParam_Input ;PLC Stn
	strcpy(ADR(SqlRequest[mySql].Parameters[0].Param_String),ADR(myPrgString))
	SqlRequest[mySql].Parameters[1].Type = cSQLParam_Input ;BatchID;
	strcpy(ADR(SqlRequest[mySql].Parameters[1].Param_String),ADR(myCatString))
	SqlRequest[mySql].Parameters[2].Type = cSQLParam_Input ; Prg
	strcpy(ADR(SqlRequest[mySql].Parameters[2].Param_String),ADR(myCusString))
ENDIF

IF SqlRequest[mySql].Complete THEN ; ClearRequest
	;Copy Out Reply Done in step.!
	SqlRequest[mySql] = cEmptySQlReq
	SqlWriteActive = FALSE
ELSE IF SqlRequest[mySql].Fail THEN
	WaitReply = FALSE ; Move to next and try and again
	SqlWriteActive = FALSE ; Reload Parameters
	SqlRequest[mySql].Fail = FALSE
;ELSE IF WaitReply AND NOT SqlWriteActive THEN
;	WaitReply = FALSE
ENDIF

END_PROGRAM
```

### Library Logical/SQL/zzSQL_Lib (IEC, version 1.00.1)
Depends on: AsDb, AsIecCon, AsTime, runtime, standard, AsString

- Program Logical/SQL/zzSQLDriver (IEC, version 1.00.1) (no source held here)

### Program Logical/SQL/zzTvText (IEC)

- Supertrack Programming Standards V1.00.1.docx (binary file, 192382 bytes)
- Standard Sequence Template.docx (binary file, 202067 bytes)
### Package Logical/BaseStandards/Alarms - A package of related programs and data objects.

### Alarms.var - Global variables
```iecst
(********************************************************************
 * COPYRIGHT -- HP
 ********************************************************************
 * Package: Alarms
 * File: Alarms.var
 * Author: treamsbottom
 * Created: March 19, 2015
 ********************************************************************
 * Variables of package Alarms
 ********************************************************************)
VAR CONSTANT
	ALM_NOALARM : UINT := 0;
	ALM_EMERGENCY_STOP : UINT := 1;
	ALM_MOTOROVERLOAD : UINT := 2;
	ALM_ULD_PROG_FINISHED : UINT := 3;
	ALM_ULD_NO_BAG : UINT := 4;
	ALM_SWITCH_FAULT : UINT := 5;
	ALM_BAG_NOT_ARRIVED : UINT := 6;
	ALM_BAG_NOT_SETTLED : UINT := 7;
	ALM_BAG_NOT_RELEASED : UINT := 9;
	ALM_LOAD_NOT_DROPPED : UINT := 10;
	ALM_CARRIAGE_MOVE_FAULT : UINT := 11;
	ALM_PHOTOCELL_BLOCKED : UINT := 12;
	ALM_PHOTOCELL_NOT_MADE : UINT := 13;
	ALM_STATION_NOT_CLOSED : UINT := 14;
	ALM_GENERAL_SEQUENCE : UINT := 15;
	ALM_BAG_NOT_AT_PROX : UINT := 16;
	ALM_BAG_NOT_SHOWN_ON_SCREEN : UINT := 17;
	ALM_INVERTOR_FAULT : UINT := 18;
	ALM_DEST_NOT_VALID : UINT := 19;
	ALM_BAG_DATA_ERROR : UINT := 20;
	ALM_BAG_OVERWEIGHT : UINT := 21;
	ALM_STATION_NOT_EMPTY : UINT := 22;
	ALM_CLEARING_BELT : UINT := 23;
	ALM_SYSTEM_STOPPED : UINT := 25;
	ALM_SWITCH_FAULT_RELEASE : UINT := 26;
	ALM_SWITCH_FAULT_RECIEVE : UINT := 27;
	ALM_RAIL_NOT_ALIGNED : UINT := 28;
	ALM_RB_LIFT_REF_NOT_FOUND : UINT := 29;
	ALM_RB_LIFT_PARAMETER_ERROR : UINT := 30;
	ALM_RB_LIFT_REF_SWITCH_FAULT : UINT := 31;
	ALM_RB_ROTATE_REF_NOT_FOUND : UINT := 32;
	ALM_RB_ROTATE_PARAMETER_ERROR : UINT := 33;
	ALM_RB_ROTATE_REF_SWITCH_FAULT : UINT := 34;
	ALM_BATCH_NO_ID_FROM_SERVER : UINT := 40;
	ALM_AIR_PRESSURE_LOW : UINT := 41;
	ALM_SEQ_DISABLED : UINT := 45;
	ALM_BACKUP_NOT_RUNNING : UINT := 50;
END_VAR
```

### Package Logical/BaseStandards/BagStacker - Bag stacker On & Off going

### Program Logical/BaseStandards/BagStacker/x_bsn (IEC, version 1.00.4) - Bag stacker ongoing

#### bsn.var - Local variables
```iecst
(********************************************************************
 * COPYRIGHT -- HP
 ********************************************************************
 * Program: 11_x_Bson
 * File: 11_x_Bson.var
 * Author: zmclaren
 * Created: May 15, 2015
 ********************************************************************
 * Local variables of program 11_x_Bson
 ********************************************************************)
VAR
	myIO : UINT;
	mySeq : UINT;
	myBS : UINT;
	myBuffBag : UINT;
	useRequest : BOOL;
	myZone : UINT;
	bsn_Enable : BOOL;
	i_bagAtBuffer : BOOL;
	i_onLineA : BOOL;
	i_tiltA : BOOL;
	i_tiltB : BOOL;
	i_bagout : BOOL;
	o_openBufferStop : BOOL;
	o_selectLineA : BOOL;
	o_selectLineB : BOOL;
	o_openStops : BOOL;
	o_tiltCylinder : BOOL;
	o_operatePusher : BOOL;
	step : UINT;
	pls : BOOL;
	lastStep : UINT;
	ton_10ms_PointReset : TON_10ms;
	ton_10ms_SettledBuffer : TON_10ms;
	ton_10ms_BagAtTilt : TON_10ms;
	ton_10ms_TiltDown : TON_10ms;
	ton_10ms_TiltUp : TON_10ms;
	ton_10ms_NotFull : TON_10ms;
	ton_10ms_Pushed : TON_10ms;
	ton_10ms_o_operatePusher : TON_10ms;
	timerAlarm : TON_10ms;
	myBag : UINT;
	bufferSettleTime : UDINT;
	releaseValid : BOOL;
	useRotary : BOOL;
	i_bagAtRotary : BOOL;
	o_openRotaryStop : BOOL;
	ton_10ms_SettledAtRotary : TON_10ms;
	settledOnRotary : BOOL;
	alarm : REFERENCE TO Alm;
	bag : REFERENCE TO Bag_typ;
	bag_buff : REFERENCE TO Bag_typ;
END_VAR
```

#### bsn.st - Implementation code
```iecst
(********************************************************************
 * COPYRIGHT -- HP
 ********************************************************************
 * Program: 11_x_Bson
 * File: 11_x_Bson.st
 * Author: zmclaren
 * Created: May 15, 2015
 ********************************************************************
 * Implementation of program 11_x_Bson
 ********************************************************************)
//V1.00.1 First Release.

PROGRAM _INIT
//Configuration
myIO				:= 231;   	//IO module number (will use 2 modules)
mySeq				:= 11;	   	//Sequence number
myBS				:= 1;	   	//Bag Stacker number
myBag				:= 0;		//
myBuffBag			:= 0;	   	//Empty bag buffer bag number - used when tracking empty bags
useRequest			:= FALSE; 	//Use the Request bit. Only use when working with x_1_point. otherwise use RequestRelease as the i_bagAtBuffer.
bufferSettleTime	:= 300;  	// Time for bag to settle at buffer in.

useRotary			:= FALSE;	// Use Rotary Point
myZone 				:= 0;

alarm						ACCESS ADR(Alarm[mySeq]);
bag							ACCESS ADR(Bag[myBag]);
bag_buff					ACCESS ADR(Bag[myBuffBag]);

END_PROGRAM

PROGRAM _CYCLIC

//IO Configuration
bsn_Enable 			:= (D[mySeq] > 0) AND NOT Std.HaltSysZone[myZone];

i_bagAtBuffer		:= X[myIO + 0].X01;
i_onLineA		  	:= X[myIO + 0].X02;
i_bagAtRotary	  	:= X[myIO + 0].X03;
i_tiltA				:= X[myIO + 1].X01;
i_tiltB				:= X[myIO + 1].X02;
i_bagout			:= X[myIO + 1].X03;

o_openBufferStop    := FALSE;
o_selectLineA		:= FALSE;
o_selectLineB		:= FALSE;
o_openStops			:= FALSE;
o_tiltCylinder		:= FALSE;
o_operatePusher		:= FALSE;
o_openRotaryStop	:= FALSE;

Request.BSN[myBS]    := FALSE;
RequestRel.BSN[myBS] := FALSE;

//Alarm
IF (myBag = 0) THEN
	alarm.Bag	:= mySeq + 10000;
ELSE
	alarm.Bag	:= myBag;
END_IF;
alarm.Name 		:= 0;
alarm.Beacon	    := TRUE;
alarm.Extra		:= 0;
alarm.Time		:= 3000;

//Setup Sequence
step := D[900 + mySeq];
//Setup Pulse contact
pls := (step <> lastStep);
lastStep := step;

//Set Sequence
IF (step = 0) THEN
	//Disabled
END_IF;

//Select Line 'A'
ton_10ms_PointReset(IN:= (step = 1), PT:= 100);
IF (step = 1) THEN
	o_selectLineA := NOT useRotary;
	IF (ton_10ms_PointReset.Q AND bsn_Enable AND NOT i_tiltA AND NOT i_tiltB AND NOT i_bagAtRotary)  THEN
		D[900 + mySeq] := 2;
		Count[mySeq] := Count[mySeq] + 1;
	END_IF;
	IF i_tiltA OR i_tiltB OR i_bagAtRotary THEN
		alarm.Name := ALM_SWITCH_FAULT;
	END_IF;
END_IF;

//Wait for bag at buffer if used
ton_10ms_SettledBuffer(IN:= i_bagAtBuffer, PT:= bufferSettleTime);
IF (step = 2) THEN
	o_selectLineA := NOT useRotary;
	IF NOT i_onLineA THEN
		IF useRequest THEN
			D[900 + mySeq] := 3;
		ELSE
			IF ton_10ms_SettledBuffer.Q THEN
				IF (myBag > 0) THEN
					IF (bag_buff.Cat > 0) AND (bag.Cat = 0) THEN
						D[900 + mySeq] := 3;
					ELSIF (bag_buff.Cat = 0) THEN
						alarm.Name := ALM_BAG_DATA_ERROR;
						alarm.Bag := myBuffBag;
					ELSE
						alarm.Name := ALM_BAG_DATA_ERROR;
					END_IF;
				ELSE
					D[900 + mySeq] := 3;
				END_IF;
			ELSIF (myBuffBag > 0) AND (bag_buff.Cat > 0) THEN
				alarm.Name := ALM_BAG_NOT_SETTLED;
			END_IF;
		END_IF;
	ELSE
		alarm.Name := ALM_SWITCH_FAULT;
		alarm.Time := 0;
	END_IF;
END_IF;

//Open buffer stop / Request bag
IF (step = 3) THEN
	releaseValid := ((myBag = 0) OR ((bag.Cat = 0) AND (bag_buff.Cat > 0)));
	o_selectLineA 	  := NOT useRotary;
	o_openRotaryStop :=	useRotary;
	o_openBufferStop   := releaseValid AND NOT useRequest;
	Request.BSN[myBS]  := releaseValid AND useRequest;
	IF i_onLineA AND releaseValid THEN
		IF (myBag > 0) THEN
			bag := bag_buff; //Clear empty buffer bag data if used
			bag_buff := Bag[0];
		END_IF;
		D[900 + mySeq] := 4;
	ELSIF (myBag > 0) THEN
		IF (bag.Cat > 0) THEN
			alarm.Name := ALM_BAG_DATA_ERROR;
			alarm.Time := 0;
		ELSIF (bag_buff.Cat = 0) THEN
			alarm.Name := ALM_BAG_DATA_ERROR;
			alarm.Bag := myBuffBag;
			alarm.Time := 0;
		ELSE
			alarm.Name  := ALM_BAG_NOT_ARRIVED;
		END_IF;
	ELSIF NOT useRequest THEN
		alarm.Name  := ALM_BAG_NOT_ARRIVED;
	END_IF;
END_IF;

//Select Line 'B' and Wait for bag in Tilt position
ton_10ms_BagAtTilt(IN:= i_tiltA AND i_tiltB, PT:= 300);
ton_10ms_SettledAtRotary(IN:= i_bagAtRotary, PT:= 300);
IF (step = 4) THEN
	IF useRotary THEN
		IF ton_10ms_SettledAtRotary.Q THEN
			settledOnRotary := TRUE;
		END_IF;
		o_openRotaryStop := NOT settledOnRotary;
		o_selectLineA := settledOnRotary;
		IF NOT settledOnRotary THEN
			alarm.Name  := ALM_SWITCH_FAULT;
		ELSE
			alarm.Name  := ALM_BAG_NOT_SETTLED;
		END_IF
	ELSE
		o_selectLineB 	   := TRUE;
		alarm.Name  := ALM_BAG_NOT_SETTLED;
	END_IF;
	o_openBufferStop   := NOT useRequest;
	IF ton_10ms_BagAtTilt.Q THEN
		D[900 + mySeq] := 5;
	END_IF;
ELSE
	settledOnRotary := FALSE;
END_IF;

//Tilt down
ton_10ms_TiltDown(IN:= (step = 5), PT:= 300);
IF (step = 5) THEN
	o_tiltCylinder := TRUE;
	IF ton_10ms_TiltDown.Q THEN
		D[900 + mySeq] := 6;
	END_IF;
END_IF;

//Tilt UP
ton_10ms_TiltUp(IN:= (step = 6), PT:= 300);
IF (step = 6) THEN
	IF ton_10ms_TiltUp.Q THEN
		D[900 + mySeq] := 7;
	END_IF;
END_IF;

//Check not full
ton_10ms_NotFull(IN:= NOT i_bagout, PT:= 300);
IF (step = 7) THEN
	IF ton_10ms_NotFull.Q THEN
		D[900 + mySeq] := 8;
	END_IF;
END_IF;

//Open stops to release bag
IF (step = 8) THEN
	o_openStops := TRUE;
	o_operatePusher := ton_10ms_o_operatePusher.Q;
	IF i_bagout THEN
		IF (myBag > 0) THEN
			bag := Bag[0];
		END_IF;
		D[900 + mySeq] := 1;
	END_IF;
	alarm.Name := ALM_BAG_NOT_RELEASED;
END_IF;

//Pusher Cylinder
ton_10ms_o_operatePusher(IN:= (step = 8) AND NOT ton_10ms_Pushed.Q, PT:= 500);
ton_10ms_Pushed(IN:= o_operatePusher, PT:= 500);

//Alarms
timerAlarm(IN := NOT pls AND (alarm.Name > 0),PT:= alarm.Time);
alarm.On := timerAlarm.Q;
alarm.ET := timerAlarm.ET;

//Outputs
Y[myIO + 0].Y05 := o_openBufferStop;
Y[myIO + 0].Y06 := o_selectLineA;
Y[myIO + 0].Y07 := o_selectLineB OR o_openRotaryStop;
Y[myIO + 0].Y08 := o_tiltCylinder;
Y[myIO + 1].Y05 := o_openStops;
Y[myIO + 1].Y06 := o_openStops;
Y[myIO + 1].Y07 := o_operatePusher;
END_PROGRAM
```

### Program Logical/BaseStandards/BagStacker/x_bsf (IEC, version 1.00.2) - Bag stacker offgoing

#### bsf.var - Local variables
```iecst
(********************************************************************
 * COPYRIGHT -- HP
 ********************************************************************
 * Program: 12_x_Bsof
 * File: 12_x_Bsof.var
 * Author: zmclaren
 * Created: June 24, 2015
 ********************************************************************
 * Local variables of program 12_x_Bsof
 ********************************************************************)
VAR
	myIO : UINT;
	mySeq : UINT;
	myBS : UINT;
	myOutBag : UINT;
	myBag : UINT;
	myUseBuff : BOOL;
	myZone : UINT;
	myRelLine : UINT;
	myBuffIO : UINT;
	i_bagAtEmptyBuffer : BOOL;
	i_emptyBagBufferOpen : BOOL;
	i_rockSepA : BOOL;
	i_rockSepB : BOOL;
	i_tiltA : BOOL;
	i_tiltB : BOOL;
	i_outLineA : BOOL;
	i_outLineB : BOOL;
	o_openRockSep : BOOL;
	o_levelCylinder : BOOL;
	o_openLineAStop : BOOL;
	o_openLineBStop : BOOL;
	o_selectLineA : BOOL;
	o_selectLineB : BOOL;
	o_select : BOOL;
	step : UINT;
	pls : BOOL;
	lastStep : UINT;
	ton_10ms_LevelClear : TON_10ms;
	ton_10ms_SettledInSeps : TON_10ms;
	ton_10ms_SettledLevel : TON_10ms;
	ton_10ms_LevellerDown : TON_10ms;
	ton_10ms_LevellerUp : TON_10ms;
	timerAlarm : TON_10ms;
	ton_10ms_PRLineClear : ARRAY[0..2] OF TON_10ms;
	bsf_Enable : BOOL;
	releaseValid : BOOL;
	useRotary : BOOL;
	i_bagAtRotary : BOOL;
	o_openRotaryStop : BOOL;
	settledOnRotary : BOOL;
	ton_10ms_SettledAtRotary : TON_10ms;
	ton_10ms_RotaryInPosition : TON_10ms;
	alarm : REFERENCE TO Alm;
	bag : REFERENCE TO Bag_typ;
	bag_out : REFERENCE TO Bag_typ;
	line_release : REFERENCE TO Line_Typ;
END_VAR
```

#### bsf.st - Implementation code
```iecst
(********************************************************************
 * COPYRIGHT -- HP
 ********************************************************************
 * Program: 12_x_Bsof
 * File: 12_x_Bsof.st
 * Author: zmclaren
 * Created: June 24, 2015
 ********************************************************************
 * Implementation of program 12_x_Bsof
 ********************************************************************)
//V1.00.1 First Release
PROGRAM _INIT
//Configuration
myIO				:= 233;   	//IO module number (will use 3 modules)
mySeq				:= 12;	  	//Sequence number
myBS				:= 1;	  	//Bag Stacker number
myBag				:= 0;		// Create bag data in stacker if tracking
myBuffIO			:= 0;     	//Empty bag buffer IO
myRelLine			:= 0;	   	//;Bag released counter number - set TO 0 TO use RequestRel / EnableRel
myOutBag			:= Line[myRelLine].LastBag;	//Empty bag buffer bag number - used when tracking empty bags

useRotary			:= FALSE;	// Use Rotary Point
myZone 				:= 0;

alarm						ACCESS ADR(Alarm[mySeq]);
bag							ACCESS ADR(Bag[myBag]);
bag_out						ACCESS ADR(Bag[myOutBag]);
line_release				ACCESS ADR(Line[myRelLine]);
END_PROGRAM
PROGRAM _CYCLIC

//Single bag buffer after Bag Stacker - enter input and output for the proximity switch and buffer stop.
i_bagAtEmptyBuffer		:= FALSE; //X[myBuffIO].X06;
i_emptyBagBufferOpen	:= FALSE; //Y[myBuffIO].Y08;

//IO Configuration
bsf_Enable			    := (D[mySeq] > 0) AND NOT Std.HaltSysZone[myZone];

i_rockSepA				:= X[myIO + 0].X01;
i_rockSepB				:= X[myIO + 0].X02;
i_tiltA					:= X[myIO + 1].X01;
i_tiltB				    := X[myIO + 1].X02;
i_outLineA				:= X[myIO + 1].X03;
i_outLineB				:= X[myIO + 2].X01;
i_bagAtRotary	  		:= X[myIO + 2].X04;

o_openRockSep			:= FALSE;
o_levelCylinder			:= FALSE;
o_openLineAStop			:= FALSE;
o_openLineBStop			:= FALSE;
o_selectLineA			:= FALSE;
o_selectLineB			:= FALSE;
o_openRotaryStop		:= FALSE;

RequestRel.BSF[myBS]	:= FALSE;

//Alarm
IF (myBag = 0) THEN
	alarm.Bag	:= mySeq + 10000;
ELSE
	alarm.Bag	:= myBag;
END_IF;

alarm.Name 		:= 0;
alarm.Beacon	    := TRUE;
alarm.Extra		:= 0;
alarm.Time		:= 3000;

//Get bag id if  creating bag data
IF (myBag > 0) AND (bag.Cat > 0) AND (bag.Bid = 0) AND (BidStn > 0) THEN
	bag.Bid := BidStn;
	BidStn := 0;
END_IF;

//Setup Sequence
step := D[900 + mySeq];
//Setup Pulse contact
pls := (step <> lastStep);
lastStep := step;

//Set Sequence
IF (step = 0) THEN
	//Disabled
END_IF;

//Check level bag clear
ton_10ms_LevelClear(IN:= NOT i_tiltA AND NOT i_tiltB,PT:= 300);
IF (step = 1) THEN
	IF (ton_10ms_LevelClear.Q AND bsf_Enable) THEN
		D[900 + mySeq] := 2;
		Count[mySeq] := Count[mySeq] + 1;
	END_IF;
	IF bsf_Enable THEN
		alarm.Name := ALM_SWITCH_FAULT;
	END_IF;
END_IF;

//Open seperators wait for bag in sep
ton_10ms_SettledInSeps(IN:= i_rockSepA AND i_rockSepB,PT:= 200);
IF (step = 2) THEN
	o_openRockSep := TRUE;
	IF ton_10ms_SettledInSeps.Q THEN
		D[900 + mySeq] := 3;
	END_IF;
	IF i_rockSepA OR i_rockSepB THEN
		alarm.Name := ALM_BAG_NOT_SETTLED;
	END_IF;
END_IF;

//Wait for bag to settle in leveller position
ton_10ms_SettledLevel(IN:= i_tiltA AND i_tiltB,PT:= 200);
IF (step = 3) THEN
	IF ton_10ms_SettledLevel.Q THEN
		IF (myBag > 0) THEN
			bag.Cat := Std.MaxCats;
			bag.Prg := Std.MaxProg;
			bag.Cus := Std.MaxCust;
		END_IF;
		D[900 + mySeq] := 4;
	END_IF;
	alarm.Name := ALM_BAG_NOT_SETTLED;
END_IF;

//Move bag leveller down
ton_10ms_LevellerDown(IN:= (step = 4),PT:= 300);
IF (step = 4) THEN
	o_levelCylinder := TRUE;
	IF ton_10ms_LevellerDown.Q THEN
		D[900 + mySeq] := 5;
	END_IF;
END_IF;

//Allow bag leveller to retract
ton_10ms_LevellerUp(IN:= (step = 5),PT:= 300);
IF (step = 5) THEN
	IF (ton_10ms_LevellerUp.Q AND NOT EnableRel.BSF[myBS]) THEN
		D[900 + mySeq] := 6;
	END_IF;
END_IF;

//Check for space on empty bag buffer / Request release
IF (step = 6) THEN
	releaseValid := (NOT i_bagAtEmptyBuffer AND NOT i_emptyBagBufferOpen AND ((myBag = 0) OR ((bag.Cat > 0) AND (bag_out.Cat = 0))));
	IF (myRelLine > 0) THEN
		IF (line_release.Clear AND releaseValid) THEN
			C[myRelLine] := 0;
			D[900 + mySeq] := 7;
		END_IF;
		IF (line_release.Clear AND i_bagAtEmptyBuffer AND NOT i_emptyBagBufferOpen) THEN
			alarm.Name := ALM_SWITCH_FAULT;
		ELSIF (myBag > 0) AND (bag.Cat = 0) THEN
			alarm.Name := ALM_BAG_DATA_ERROR;
			alarm.Time := 0;
		ELSIF line_release.Clear AND (myOutBag > 0) AND (bag_out.Cat > 0) THEN
			alarm.Name := ALM_BAG_DATA_ERROR;
			alarm.Bag := myOutBag;
			alarm.Time := 0;
		END_IF;
	ELSE
		RequestRel.BSF[myBS] := releaseValid;
		IF EnableRel.BSF[myBS] AND releaseValid THEN
			D[900 + mySeq] := 7;
		ELSIF (myBag > 0) AND (bag.Cat = 0) THEN
			alarm.Name := ALM_BAG_DATA_ERROR;
			alarm.Time := 0;
		ELSIF (myOutBag > 0) AND (bag_out.Cat > 0) THEN
			alarm.Name := ALM_BAG_DATA_ERROR;
			alarm.Bag := myOutBag;
			alarm.Time := 0;
		END_IF;
	END_IF;
END_IF;

//Open stop on line 'A'
IF (step = 7) THEN
	o_openLineAStop := TRUE;
	o_selectLineA	:= TRUE;
	IF i_outLineA THEN
		D[900 + mySeq] := 8;
	END_IF;
	alarm.Name := ALM_BAG_NOT_RELEASED;
END_IF;

//Open stop on line 'B'
IF (step = 8) THEN
	o_openLineBStop := TRUE;
	o_selectLineA	:= TRUE;
	IF i_outLineB THEN
		D[900 + mySeq] := 9;
	END_IF;
	alarm.Name := ALM_BAG_NOT_RELEASED;
END_IF;

//Select bag stop and wait for bag out of leveller
ton_10ms_SettledAtRotary(IN:= i_bagAtRotary, PT:= 300);
ton_10ms_RotaryInPosition(IN:= settledOnRotary, PT:= 200);
IF (step = 9) THEN
	IF useRotary THEN
		IF ton_10ms_SettledAtRotary.Q THEN
			settledOnRotary := TRUE;
		END_IF;
		o_selectLineA := NOT settledOnRotary;
		o_openRotaryStop := ton_10ms_RotaryInPosition.Q;
		IF NOT settledOnRotary THEN
			alarm.Name  := ALM_SWITCH_FAULT;
		END_IF
	ELSE
		o_selectLineB := TRUE;
	END_IF;
	IF (myBag = 0) THEN
		IF (myRelLine > 0) THEN
			IF line_release.Trip THEN
				D[900 + mySeq] := 1;
			END_IF;
		ELSE
			IF NOT EnableRel.BSF[myBS] THEN
				D[900 + mySeq] := 1;
			END_IF;
		END_IF;
		alarm.Name := ALM_BAG_NOT_RELEASED;
	ELSE//Use tracking
		IF (myRelLine > 0) THEN
			IF line_release.Trip AND (bag.Cat > 0) AND (bag_out.Cat = 0) THEN
				bag_out := bag;
				bag := Bag[0];
				D[900 + mySeq] := 1;
			END_IF;
		ELSE
			IF NOT EnableRel.BSF[myBS] AND (bag.Cat = 0) THEN // Make sure data is copied out by enabling sequence.
				D[900 + mySeq] := 1;
			ELSIF NOT EnableRel.BSF[myBS] AND (bag.Cat > 0) THEN
				alarm.Name := ALM_BAG_DATA_ERROR;
			END_IF;
		END_IF;
	END_IF;
ELSE
	settledOnRotary := FALSE;
END_IF;

//Alarms
timerAlarm(IN := NOT pls AND (alarm.Name > 0),PT:= alarm.Time);
alarm.On := timerAlarm.Q;
alarm.ET := timerAlarm.ET;

//SBS Offgoing Bagstacker Pressure relief
ton_10ms_PRLineClear[0](IN:= (NOT X[myIO + 0].X03 AND NOT X[myIO + 0].X04),PT:= 500);
Y[myIO + 0].Y07 := ton_10ms_PRLineClear[0].Q;

//Outputs
Y[myIO + 0].Y05 := o_openRockSep;
Y[myIO + 0].Y06 := o_openRockSep;
Y[myIO + 1].Y05 := o_openLineAStop;
Y[myIO + 1].Y06 := o_openLineBStop;
Y[myIO + 1].Y07 := o_levelCylinder;
Y[myIO + 2].Y05 := o_selectLineA;
Y[myIO + 2].Y06 := o_selectLineB OR o_openRotaryStop;
END_PROGRAM
```

- Standard Sequence bsf ENG.docx (binary file, 206090 bytes)
- Standard Sequence bsn ENG.docx (binary file, 206437 bytes)
### Package Logical/BaseStandards/Discharger - Discharger with Batching options

### Program Logical/BaseStandards/Discharger/x_dc (IEC, version 1.00.1) - Discharger

#### x_dc.var - Local variables
```iecst
(********************************************************************
 * COPYRIGHT -- HP
 ********************************************************************
 * Program: 6_x_Dc
 * File: 6_x_Dc.var
 * Author: zmclaren
 * Created: May 14, 2015
 ********************************************************************
 * Local variables of program 6_x_Dc
 ********************************************************************)
VAR
	myIO : UINT;
	myStartStop : UINT;
	mySeq : UINT;
	myDC : UINT;
	myBuffBag : UINT;
	myBag : UINT;
	myDst : USINT;
	myZone : UINT;
	myBagCloser : BOOL;
	myCodesStrobe : BOOL;
	myPushButtonControl : BOOL;
	myPickerControl : BOOL;
	myCan : UINT;
	i_bagAtEmptyBuffer : BOOL;
	o_emptyBagBufferOpen : BOOL;
	i_bagAtBuffer : BOOL;
	i_bagAtDischarger : BOOL;
	i_openBag : BOOL;
	i_loadDropped : BOOL;
	i_bagReleased : BOOL;
	i_bagEmpty : BOOL;
	o_bagReady : BOOL;
	o_openBuffer : BOOL;
	o_steadys : BOOL;
	o_closer : BOOL;
	o_openBag : BOOL;
	o_openStop : BOOL;
	step : UINT;
	pls : BOOL;
	lastStep : UINT;
	myDCBatch : BOOL;
	n : UINT;
	ton_10ms_SettledBuffer : TON_10ms;
	ton_10ms_SettledAtDischarger : TON_10ms;
	ton_10ms_SteadysDown : TON_10ms;
	ton_10ms_MinOpen : TON_10ms;
	ton_10ms_CloserDown : TON_10ms;
	ton_10ms_CloserUp : TON_10ms;
	ton_10ms_SteadyUp : TON_10ms;
	timerAlarm : TON_10ms;
	dischargerEnable : BOOL;
	batchSizeSet : UINT;
	batchWeightSet : UINT;
	matchCus : BOOL;
	temp_BatchSize : UINT;
	searchDepth : UINT;
	useBuffer : BOOL;
	TestDischarger : BOOL;
	LoadDropped : BOOL;
	TestDrop : BOOL;
	UseCounter : BOOL;
	ton_10ms_CloserDelay : TON_10ms;
	ExitLoop : BOOL;
	BatchValue : UINT;
	CodeStep : BOOL;
	alarm : REFERENCE TO Alm;
	myRelLine : UINT;
	bag : REFERENCE TO Bag_typ;
	bag_buff : REFERENCE TO Bag_typ;
	bag_out : REFERENCE TO Bag_typ;
	can : REFERENCE TO CAN_Vars;
	line_release : REFERENCE TO Line_Typ;
END_VAR
```

#### x_dc.st - Implementation code
```iecst
(********************************************************************
 * COPYRIGHT -- HP
 ********************************************************************
 * Program: 6_x_Dc
 * File: 6_x_Dc.st
 * Author: zmclaren
 * Created: May 14, 2015
 ********************************************************************
 * Implementation of program 6_x_Dc
 ********************************************************************)
//Version 1.00.0 First Release.

PROGRAM _INIT
//Configuration
myIO					:= 151;   //Discharger IO module number
myStartStop				:= 6;     //Start / Stop used on TrackView display (Traffic Light)
mySeq					:= 6;     //Sequence number
myDC					:= 1;     //Discharger number
myCan					:= 1;     //Discharger CAN / KanLink as may differ from discharger number
myBuffBag				:= 251;   //Buffer bag number - set to 0 to use Request / Enable
myBag					:= 151;   //Discharger bag number
myDst					:= 11;    //Destination number for bags to be opened at this discharger (destination 0 will also be opened)
myRelLine				:= 0;     //Bag released counter number - set to 0 to use RequestRel / EnableRel
myZone					:= 0;     //Safe Zone

myBagCloser				:= TRUE;  //Bag closer is fitted?
myCodesStrobe			:= FALSE; //Use Jensen (Senking) strobe method for transfer of codes to CBW
myPushButtonControl		:= FALSE; //Bag is opened by pressing a pushbutton and confirmed empty with a second press.
myPickerControl			:= FALSE; //Bag is opened by a picker (only open bag signal which goes off when load has dropped)
//Batching controls Kanlink Only....
myDCBatch               := FALSE; //Use batch for Kan link
batchSizeSet 			:= 980; // D Registers.
batchWeightSet 			:= 981;
matchCus 				:= TRUE;

alarm						ACCESS ADR(Alarm[mySeq]);
bag							ACCESS ADR(Bag[myBag]);
bag_buff					ACCESS ADR(Bag[myBuffBag]);
can							ACCESS ADR(CAN[myCan]);
line_release				ACCESS ADR(Line[myRelLine]);

END_PROGRAM

PROGRAM _CYCLIC

IF myPushButtonControl OR myPickerControl THEN
	can.DropLoad		:= X[0].X01; //Input open bag
    can.LoadDropped	:= X[0].X02; //Input load has dropped if used
END_IF;

//Single bag buffer after discharger - enter input and output for the proximity switch and buffer stop.
i_bagAtEmptyBuffer		:= FALSE;
o_emptyBagBufferOpen	:= FALSE;

//IO Configuration

dischargerEnable 		:= ((D[myStartStop] > 0) AND NOT Std.HaltSysZone[myZone]);

i_bagAtBuffer			:= X[myIO].X01;
i_bagAtDischarger		:= X[myIO].X02;
i_openBag				:= can.DropLoad;
i_loadDropped			:= can.LoadDropped;
i_bagReleased			:= X[myIO].X03;
i_bagEmpty			  	:= X[myIO].X04;

o_bagReady				:= FALSE;
o_openBuffer 			:= FALSE;
o_steadys				:= FALSE;
o_closer				:= FALSE;
o_openBag				:= FALSE;
o_openStop				:= FALSE;

Request.DC[myDC]		:= FALSE;
RequestRel.DC[myDC] 	:= FALSE;

//Setup Alarm
IF (myBag = 0) THEN
	alarm.Bag	:= mySeq + 10000;
ELSE
	alarm.Bag	:= myBag;
END_IF;
alarm.Name 		:= 0;
alarm.Beacon	    := TRUE;
alarm.Extra		:= 0;
alarm.Time		:= 3000;

//Setup Sequence
step := D[900 + mySeq];
//Setup Pulse contact
pls := (step <> lastStep);
lastStep := step;

//Set Sequence
IF (step = 0) THEN
	//Disabled
END_IF;

//*************************************************Batch Calculation**************************************************************
IF myDCBatch THEN

	batchSizeSet	:= D[2800 + bag_buff.Prg];

	//Calculate buffer data to send to PT - note even 2nd bag of batch will have different weight.
	IF (step = 1) AND (batchSizeSet > 1) AND (bag_buff.Cat > 0) THEN
		//Error Protection
		IF (D[batchSizeSet] > batchSizeSet) THEN	 //If we get a data reg error then recalculate.
			D[batchSizeSet] := 0;
		END_IF;
		FOR n := 0 TO 5 DO
			can.Batchpart[n].Customer := 0;
			can.Batchpart[n].Wgt := 0;
		END_FOR;
		D[batchWeightSet] := bag_buff.Wgt;
		can.Batchpart[0].Customer := bag_buff.Cus;
		can.Batchpart[0].Wgt := bag_buff.Wgt;
		temp_BatchSize := 1;
		ExitLoop := FALSE;

		IF (D[batchSizeSet] < 1) THEN
			BatchValue := batchSizeSet;
		ELSE
			BatchValue	:= D[batchSizeSet];
		END_IF;
		IF (BatchValue > 1) THEN
			searchDepth := 0;
			FOR n := 1 TO (BatchValue - 1)DO
				IF (Bag[myBuffBag + n].Cat > 0) THEN
					searchDepth := n + 1; // Add 1 to allow for position 0
				END_IF;
				IF ((Bag[myBuffBag + n].Cat = bag_buff.Cat) AND ((Bag[myBuffBag + n].Cus = bag_buff.Cus) OR NOT matchCus))THEN
					D[batchWeightSet] := D[batchWeightSet] + Bag[myBuffBag + n].Wgt; // Sum Wieghts
					can.Batchpart[n].Customer := Bag[myBuffBag + n].Cus;
					can.Batchpart[n].Wgt := Bag[myBuffBag + n].Wgt;
					temp_BatchSize := n + 1;
				ELSE
					ExitLoop := TRUE;
				END_IF;
				IF ExitLoop THEN
					EXIT;
				END_IF;
			END_FOR;
			IF (D[batchSizeSet] = 0) AND ((temp_BatchSize = batchSizeSet) OR (searchDepth >= batchSizeSet)) THEN	// Check we have searched all bags required.
				D[batchSizeSet] := temp_BatchSize;
			END_IF;
		END_IF;
	ELSE IF (step = 1) AND (batchSizeSet <= 1) AND (bag_buff.Cat > 0) THEN
			D[batchSizeSet] := 1;
			D[batchWeightSet] := bag_buff.Wgt;
			can.Batchpart[0].Customer := bag_buff.Cus;
			can.Batchpart[0].Wgt := bag_buff.Wgt;
		END_IF;
	END_IF;
 	can.Batch_QtyRemaining := D[batchSizeSet];
ELSE
	can.Batch_QtyRemaining := 0;
END_IF;

//*******************************************************END BATCHING CALC****** SEE step 6 from Batch decrement**********************************

//Check Status - Bag settled at buffer, no bag at discharger, bag at buffer on screen and no bag at discharger on the screen
useBuffer := (myBuffBag > 0);
ton_10ms_SettledBuffer(IN:= i_bagAtBuffer, PT:= 300);
IF (step = 1) THEN
	//Disable sequence if input made
	IF (dischargerEnable AND NOT i_bagAtDischarger AND (bag.Cat = 0) AND NOT Std.HaltSysZone[myZone]) THEN
		IF useBuffer AND NOT myDCBatch THEN  // No batch standerd
			IF (ton_10ms_SettledBuffer.Q AND (bag_buff.Cat > 0)) THEN
				D[900 + mySeq] := 2;
				Count[mySeq] := Count[mySeq] + 1;
			END_IF;
		ELSIF useBuffer AND myDCBatch THEN  // Use Batch set myDCBatch
			IF (ton_10ms_SettledBuffer.Q AND (bag_buff.Cat > 0) AND (D[batchSizeSet] > 0)) THEN // Make sure batch size has arrived in buffer.
				D[900 + mySeq] := 2;
				Count[mySeq] := Count[mySeq] + 1;
			END_IF;

			//Alarm - Buffer bag detection error
			IF (myBuffBag > 0) THEN
				IF (bag_buff.Cat > 0) AND NOT i_bagAtBuffer THEN
					alarm.Name 	:= almBagNotAtProx;
					alarm.Bag	:= myBuffBag;
				ELSIF  (bag_buff.Cat = 0) AND i_bagAtBuffer THEN
					alarm.Name 	:= almBagNotShownOnScreen;
					alarm.Bag	:= myBuffBag;
				END_IF;
			END_IF;
		ELSE
			D[900 + mySeq] := 2;
			Count[mySeq] := Count[mySeq] + 1;
		END_IF;
	END_IF;

	//Alarm - Bag detected at discharger
	IF (bag.Cat > 0) THEN
		alarm.Name := almBagDataError;
	ELSIF i_bagAtDischarger THEN
		alarm.Name := almSwitchFault;
	END_IF;
END_IF;

//Wait for bag in discharger
IF (step = 2) THEN
	o_openBuffer 		:= useBuffer;
	Request.DC[myDC] 	:= NOT useBuffer;
	IF i_bagAtDischarger THEN
		D[900 + mySeq] := 3;
	END_IF;
	IF useBuffer THEN
		alarm.Name := almBagNotArrived;
	END_IF;
END_IF;

//Let bag settle in discharger
ton_10ms_SettledAtDischarger(IN:= i_bagAtDischarger, PT:= 300);
IF (step = 3) THEN
	IF useBuffer THEN
		IF ((bag.Cat = 0) AND (bag_buff.Cat > 0)) THEN
			bag 		:= bag_buff;
			bag_buff 	:= Bag[0];
		END_IF;
	END_IF;
	IF ((bag.Dst <> myDst) AND (bag.Dst <> 0)) THEN
		D[900 + mySeq] := 11; //Bag is for another destination then go-to release bag
	END_IF;
	IF ton_10ms_SettledAtDischarger.Q AND i_bagEmpty THEN  //Make sure empty bag photocell is working (Cannot be set to NOT at top)
		D[900 + mySeq] := 4;
	END_IF;
	alarm.Name := almBagNotSettled;
END_IF;

//Allow steadys to move down
ton_10ms_SteadysDown(IN:= (step = 4), PT:= 300);
IF (step = 4) THEN
	IF ton_10ms_SteadysDown.Q THEN
		IF (bag.Prg = Std.MaxProg) THEN
			D[900 + mySeq] := 8; //Empty bag then go-to close
		ELSE
			IF myCodesStrobe THEN
				IF can.StrobeComplete THEN
					D[900 + mySeq] := 5;
				END_IF
			ELSIF myPushButtonControl THEN
				IF NOT i_openBag THEN
					D[900 + mySeq] := 5;
				END_IF;
				alarm.Name := almSwitchFault;
			ELSE
				D[900 + mySeq] := 5;
			END_IF;
		END_IF;
	END_IF;
END_IF;

//Steady cylinders on from steps 4 - 9
o_steadys := ((step >= 4) AND (step <= 9));

//Bag opener on from step 5 - 8
o_openBag := ((step >= 6) AND (step <= 8));

CodeStep  := ((step >= 5) AND (step <= 6));

//Wash Codes
IF CodeStep THEN
	can.Program		:= bag.Prg;
	can.Category 	:= bag.Cat;
	can.Customer 	:= bag.Cus;
	can.Weight   	:= bag.Wgt;   //D[batchWeightSet] (WgtRound / 10) ;rounded up weight divide BY 10
	can.BatchID		:= bag.Mis;
	can.DoubleLoad 	:= FALSE;
ELSE
	can.Program 		:= 0;
	can.Category 	:= 0;
	can.Customer 	:= 0;
	can.Weight   	:= 0;
	can.BatchID		:= 0;
	can.DoubleLoad 	:= FALSE;
END_IF;

//Bag Ready to Washing Machine
IF (step = 5) THEN
	o_bagReady 			:= myPushButtonControl OR myPickerControl;
	can.BagReady := NOT myPushButtonControl OR myPickerControl;
	IF i_openBag OR TestDischarger THEN
		D[900 + mySeq] := 6;
	END_IF;
ELSE
	can.BagReady	:= FALSE;
END_IF;

//Set LoadDropped to False
IF (step <> 6) THEN
	LoadDropped := FALSE;
END_IF;

//Open Bag Until LoadDropped Received and has been open for 6 seconds
ton_10ms_MinOpen(IN:= (step = 6), PT:= 600);
IF (step = 6) THEN

	IF (myPushButtonControl OR myPickerControl) THEN
		IF (NOT i_openBag OR TestDischarger) THEN
			LoadDropped := TRUE;
		END_IF;
	ELSE
		IF (i_loadDropped OR TestDischarger) THEN
			LoadDropped := TRUE;
		END_IF;
	END_IF;

	IF (LoadDropped AND ton_10ms_MinOpen.Q) THEN
		//Write Report
		IF (ReportUnloading[myDC].Cat = 0) THEN
			ReportUnloading[myDC].Prg := bag.Prg; 	//Program
			ReportUnloading[myDC].Cat := bag.Cat;	//Category
			ReportUnloading[myDC].Cus := bag.Cus;	//Customer
			ReportUnloading[myDC].Wgt := bag.Wgt;	//Weight
			ReportUnloading[myDC].Cnt := 0;					//Count
			ReportUnloading[myDC].Stn := 0;					//Station
			ReportUnloading[myDC].Mcn := myDC;				//Machine
			ReportUnloading[myDC].Mis := bag.Mis;	//Batch ID
			IF (batchSizeSet > 0) AND (D[batchSizeSet] > 0)  THEN D[batchSizeSet] := (D[batchSizeSet] - 1); END_IF;
			D[900 + mySeq] := 7;
		END_IF;
	END_IF;
	alarm.Time := 3000;
	alarm.Name := almLoadNotDropped;
END_IF;

//Change display to empty bag - clear all other bag data
IF (step = 7) THEN
	IF myPushButtonControl THEN
		o_bagReady := Std.Clock200ms;
		IF ((i_openBag AND NOT i_loadDropped AND NOT i_bagEmpty) OR TestDrop) THEN
			bag		:= Bag[0];
			bag.Prg 	:= Std.MaxProg;
			bag.Cat	:= Std.MaxCats;
			D[900 + mySeq] 	:= 8;
		END_IF;
		IF (i_loadDropped OR i_bagEmpty) THEN
			alarm.Name := almSwitchFault;
		END_IF;
	ELSE
		IF ((NOT i_openBag AND NOT i_loadDropped AND NOT i_bagEmpty) OR TestDrop) THEN
			bag		:= Bag[0];
			bag.Prg 	:= Std.MaxProg;
			bag.Cat	:= Std.MaxCats;
			D[900 + mySeq] 	:= 8;
		END_IF;
		IF (i_openBag OR i_loadDropped OR i_bagEmpty) THEN
			alarm.Name := almSwitchFault;
		END_IF;
	END_IF;
END_IF;

//Close bag
ton_10ms_CloserDelay(IN:= (step = 8), PT:= 200);
ton_10ms_CloserDown(IN:= (step = 8), PT:= 800);
IF (step = 8) THEN
	IF myBagCloser THEN
		o_closer := ton_10ms_CloserDelay.Q;
		IF ton_10ms_CloserDown.Q THEN
			D[900 + mySeq] := 9;
		END_IF;
	ELSE
		D[900 + mySeq] := 10;
	END_IF;
END_IF;

//Allow closer to go back up
ton_10ms_CloserUp(IN:= (step = 9), PT:= 600);
IF (step = 9) THEN
	IF ton_10ms_CloserUp.Q THEN
		D[900 + mySeq] := 10;
	END_IF;
END_IF;

//Allow steadys to go up
ton_10ms_SteadyUp(IN:= (step = 10), PT:= 200);
IF (step = 10) THEN
	IF ton_10ms_SteadyUp.Q AND NOT EnableRel.DC[myDC] THEN
		D[900 + mySeq] := 11;
	END_IF;
END_IF;

//Check for space on empty bag buffer / Request release
UseCounter := (myRelLine > 0);
IF (step = 11) THEN
	IF UseCounter THEN
		IF (line_release.Clear AND NOT i_bagAtEmptyBuffer AND NOT o_emptyBagBufferOpen) THEN
			D[900 + mySeq] := 12;
		END_IF;
		IF (line_release.Clear AND i_bagAtEmptyBuffer AND NOT o_emptyBagBufferOpen) THEN
			alarm.Name := almSwitchFault;
		END_IF;
	ELSE
		RequestRel.DC[myDC]	:= TRUE;
		IF EnableRel.DC[myDC] THEN
			D[900 + mySeq] := 12;
		END_IF;
	END_IF;
END_IF;

//Open buffer stop - unitl bag out
IF (step = 12) THEN
	o_openStop := TRUE;
	bag := Bag[0]; //Clear bag;

	IF UseCounter THEN
		IF pls THEN
			C[myRelLine] := 0;
		END_IF;
		IF line_release.Trip OR i_bagReleased THEN
			D[900 + mySeq] := 1;
		END_IF;
	ELSE
		IF NOT EnableRel.DC[myDC] THEN
			D[900 + mySeq] := 1;
		END_IF;
	END_IF;
	alarm.Name := almBagNotReleased;
END_IF;

//Alarms
timerAlarm(IN := NOT pls AND (alarm.Name > 0),PT:= alarm.Time);
alarm.On 	:= timerAlarm.Q;
alarm.ET 	:= timerAlarm.ET;

//Outputs
Y[0].Y01 		:= o_bagReady;
Y[myIO].Y01 	:= o_openBuffer;
Y[myIO].Y02 	:= o_steadys;
Y[myIO].Y03 	:= o_openBag;
Y[myIO].Y04 	:= o_openStop;
Y[myIO].Y05 	:= o_closer;
END_PROGRAM
```

- Sequence_DCwithSB.doc (binary file, 82944 bytes)
### Program Logical/BaseStandards/Discharger/withStaticBag/x_dc (IEC, version 1.00.2) - *Discharger to work with Static Bag

#### x_dc.var - Local variables
```iecst
(********************************************************************
 * COPYRIGHT -- HP
 ********************************************************************
 * Program: 6_x_Dc
 * File: 6_x_Dc.var
 * Author: zmclaren
 * Created: May 14, 2015
 ********************************************************************
 * Local variables of program 6_x_Dc
 ********************************************************************)
VAR
	myIO : UINT;
	myStartStop : UINT;
	mySeq : UINT;
	myDC : UINT;
	myBuffBag : UINT;
	myBag : UINT;
	myDst : USINT;
	myRelCounter : UINT;
	myZone : UINT;
	myBagCloser : BOOL;
	myCodesStrobe : BOOL;
	myPushButtonControl : BOOL;
	myPickerControl : BOOL;
	myCan : UINT;
	i_bagAtEmptyBuffer : BOOL;
	o_emptyBagBufferOpen : BOOL;
	i_bagAtBuffer : BOOL;
	i_bagAtDischarger : BOOL;
	i_openBag : BOOL;
	i_loadDropped : BOOL;
	i_bagReleased : BOOL;
	i_bagEmpty : BOOL;
	o_bagReady : BOOL;
	o_openBuffer : BOOL;
	o_steadys : BOOL;
	o_closer : BOOL;
	o_openBag : BOOL;
	o_openStop : BOOL;
	step : UINT;
	pls : BOOL;
	lastStep : UINT;
	myDCBatch : BOOL;
	n : UINT;
	ton_10ms_SettledBuffer : TON_10ms;
	ton_10ms_SettledAtDischarger : TON_10ms;
	ton_10ms_SteadysDown : TON_10ms;
	ton_10ms_MinOpen : TON_10ms;
	ton_10ms_CloserDown : TON_10ms;
	ton_10ms_CloserUp : TON_10ms;
	ton_10ms_SteadyUp : TON_10ms;
	timerAlarm : TON_10ms;
	dischargerEnable : BOOL;
	batchSizeSet : UINT;
	batchWeightSet : UINT;
	matchCus : BOOL;
	temp_BatchSize : UINT;
	searchDepth : UINT;
	useBuffer : BOOL;
	ExitLoop : BOOL;
	BatchValue : UINT;
	CodeStep : BOOL;
	TestDischarger : BOOL;
	LoadDropped : BOOL;
	TestDrop : BOOL;
	UseCounter : BOOL;
	alarm : REFERENCE TO Alm;
	ton_10ms_CloserDelay : TON_10ms;
	myOutBag : UINT;
	outBag : REFERENCE TO Bag_typ;
	bag : REFERENCE TO Bag_typ;
	bagsPassThroughDC : BOOL;
END_VAR
```

#### x_dc.st - Implementation code
```iecst
(********************************************************************
 * COPYRIGHT -- HP
 ********************************************************************
 * Program: 6_x_Dc
 * File: 6_x_Dc.st
 * Author: zmclaren
 * Created: May 14, 2015
 ********************************************************************
 * Implementation of program 6_x_Dc
 ********************************************************************)
//Version 1.00.0 First Release.
//Version 1.00.2 Make  Can.BagReady Optional to avoid overwriting the static bag
PROGRAM _INIT
//Configuration
myIO					:= 151;   //Discharger IO module number
myStartStop				:= 6;     //Start / Stop used on TrackView display (Traffic Light)
mySeq					:= 6;     //Sequence number
myDC					:= 1;     //Discharger number
myCan					:= 0;     //Discharger CAN / KanLink as may differ from discharger number
myBuffBag				:= 0;   //Buffer bag number - set to 0 to use Request / Enable
myBag					:= 135;   //Discharger bag number
myDst					:= 21;    //Destination number for bags to be opened at this discharger (destination 0 will also be opened)
myRelCounter			:= 22;    //Bag released counter number - set to 0 to use RequestRel / EnableRel
myOutBag				:= Line[myRelCounter].LastBag; // For tracking full bags
myZone					:= 0;     //Safe Zone
myBagCloser				:= TRUE;  //Bag closer is fitted?
myCodesStrobe			:= FALSE; //Use Jensen (Senking) strobe method for transfer of codes to CBW
myPushButtonControl		:= TRUE; //Bag is opened by pressing a pushbutton and confirmed empty with a second press.
myPickerControl			:= FALSE; //Bag is opened by a picker (only open bag signal which goes off when load has dropped)
bagsPassThroughDC		:= TRUE; // Bags with different destination are allowed to pass through the discharger.

alarm					ACCESS ADR(Alarm[mySeq]);
bag						ACCESS ADR(Bag[myBag]);
outBag					ACCESS ADR(Bag[myOutBag]);

END_PROGRAM

PROGRAM _CYCLIC

IF myPushButtonControl OR myPickerControl THEN
	CAN[myCan].DropLoad		:= X[0].X01; //Input open bag
    CAN[myCan].LoadDropped	:= X[0].X02; //Input load has dropped if used
END_IF;

//Single bag buffer after discharger - enter input and output for the proximity switch and buffer stop.
i_bagAtEmptyBuffer		:= FALSE;
o_emptyBagBufferOpen	:= FALSE;

//IO Configuration

dischargerEnable 		:= ((D[myStartStop] > 0) AND NOT Std.HaltSysZone[myZone]);

i_bagAtBuffer			:= X[myIO].X01;
i_bagAtDischarger		:= X[myIO].X02;
i_openBag				:= Enable.SK[myDC];
i_loadDropped			:= FALSE;
i_bagReleased			:= X[myIO].X03;
i_bagEmpty			  	:= X[myIO].X04;  //  Do not set as NOT or False needs to be seen on step 3

o_bagReady				:= FALSE;
o_openBuffer 			:= FALSE;
o_steadys				:= FALSE;
o_closer				:= FALSE;
o_openBag				:= FALSE;
o_openStop				:= FALSE;

Request.DC[myDC]		:= FALSE;
RequestRel.DC[myDC] 	:= FALSE;

//Setup Alarm
IF (myBag = 0) THEN
	alarm.Bag	:= mySeq + 10000;
ELSE
	alarm.Bag	:= myBag;
END_IF;
alarm.Name 		:= 0;
alarm.Beacon	    := TRUE;
alarm.Extra		:= 0;
alarm.Time		:= 3000;

//Setup Sequence
step := D[900 + mySeq];
//Setup Pulse contact
pls := (step <> lastStep);
lastStep := step;

//Set Sequence
IF (step = 0) THEN
	//Disabled
END_IF;

//Check Status - Bag settled at buffer, no bag at discharger, bag at buffer on screen and no bag at discharger on the screen
useBuffer := (myBuffBag > 0);
ton_10ms_SettledBuffer(IN:= i_bagAtBuffer, PT:= 300);
IF (step = 1) THEN
	//Disable sequence if input made
	IF (dischargerEnable AND NOT i_bagAtDischarger AND (bag.Cat = 0) AND NOT Std.HaltSysZone[myZone]) THEN
		IF useBuffer AND NOT myDCBatch THEN  // No batch standerd
			IF (ton_10ms_SettledBuffer.Q AND (Bag[myBuffBag].Cat > 0)) THEN
				D[900 + mySeq] := 2;
				Count[mySeq] := Count[mySeq] + 1;
			END_IF;
		ELSIF useBuffer AND myDCBatch THEN  // Use Batch set myDCBatch
			IF (ton_10ms_SettledBuffer.Q AND (Bag[myBuffBag].Cat > 0) AND (D[batchSizeSet] > 0)) THEN // Make sure batch size has arrived in buffer.
				D[900 + mySeq] := 2;
				Count[mySeq] := Count[mySeq] + 1;
			END_IF;

			//Alarm - Buffer bag detection error
			IF (myBuffBag > 0) THEN
				IF (Bag[myBuffBag].Cat > 0) AND NOT i_bagAtBuffer THEN
					alarm.Name 	:= almBagNotAtProx;
					alarm.Bag	:= myBuffBag;
				ELSIF  (Bag[myBuffBag].Cat = 0) AND i_bagAtBuffer THEN
					alarm.Name 	:= almBagNotShownOnScreen;
					alarm.Bag	:= myBuffBag;
				END_IF;
			END_IF;
		ELSE
			D[900 + mySeq] := 2;
			Count[mySeq] := Count[mySeq] + 1;
		END_IF;
	END_IF;

	//Alarm - Bag detected at discharger
	IF (bag.Cat > 0) THEN
		alarm.Name := almBagDataError;
	ELSIF i_bagAtDischarger THEN
		alarm.Name := almSwitchFault;
	END_IF;
END_IF;

//Wait for bag in discharger
IF (step = 2) THEN
	o_openBuffer 		:= useBuffer;
	Request.DC[myDC] 	:= NOT useBuffer;
	IF i_bagAtDischarger THEN
		D[900 + mySeq] := 3;
	END_IF;
	IF useBuffer THEN
		alarm.Name := almBagNotArrived;
	END_IF;
END_IF;

//Let bag settle in discharger
ton_10ms_SettledAtDischarger(IN:= i_bagAtDischarger, PT:= 300);
IF (step = 3) THEN
	IF useBuffer THEN
		IF ((bag.Cat = 0) AND (Bag[myBuffBag].Cat > 0)) THEN
			bag := Bag[myBuffBag];
			Bag[myBuffBag] 	:= Bag[0];
		END_IF;
	END_IF;
	IF ((bag.Dst <> myDst) AND (bag.Dst <> 0)) THEN
		D[900 + mySeq] := 11; //Bag is for another destination then go-to release bag
	END_IF;
	IF ton_10ms_SettledAtDischarger.Q THEN
		IF bag.Cat = Std.MaxCats THEN
			D[900 + mySeq] := 8;
		ELSIF ((bag.Dst <> myDst) AND (bag.Dst <> 0) AND bagsPassThroughDC ) THEN
			D[900 + mySeq] := 11; //Bag is for another destination then go-to release bag
		ELSIF i_bagEmpty THEN  //Make sure empty bag photocell is working (Cannot be set to NOT at top)
			D[900 + mySeq] := 4;
		END_IF;
	ELSE
		alarm.Name := almBagNotSettled;
	END_IF;
END_IF;

//Allow steadys to move down
ton_10ms_SteadysDown(IN:= (step = 4), PT:= 300);
IF (step = 4) THEN
	IF ton_10ms_SteadysDown.Q THEN
		IF (bag.Prg = Std.MaxProg) THEN
			D[900 + mySeq] := 8; //Empty bag then go-to close
		ELSE
			IF myCodesStrobe THEN
				IF CAN[myCan].StrobeComplete THEN
					D[900 + mySeq] := 5;
				END_IF
			ELSIF myPushButtonControl THEN
				IF NOT i_openBag THEN
					D[900 + mySeq] := 5;
				END_IF;
				alarm.Name := almSwitchFault;
			ELSE
				D[900 + mySeq] := 5;
			END_IF;
		END_IF;
	END_IF;
END_IF;

//Steady cylinders on from steps 4 - 9
o_steadys := ((step >= 4) AND (step <= 9));

//Bag opener on from step 5 - 8
o_openBag := ((step >= 6) AND (step <= 8));

CodeStep  := ((step >= 5) AND (step <= 6));

////Wash Codes
//IF CodeStep THEN
//	CAN[myCan].Program		:= bag.Prg;
//	CAN[myCan].Category 	:= bag.Cat;
//	CAN[myCan].Customer 	:= bag.Cus;
//	CAN[myCan].Weight   	:= bag.Wgt;   //D[batchWeightSet] (WgtRound / 10) ;rounded up weight divide BY 10
//	CAN[myCan].BatchID		:= bag.Mis;
//	CAN[myCan].DoubleLoad 	:= FALSE;
//ELSE
//	CAN[myCan].Program 		:= 0;
//	CAN[myCan].Category 	:= 0;
//	CAN[myCan].Customer 	:= 0;
//	CAN[myCan].Weight   	:= 0;
//	CAN[myCan].BatchID		:= 0;
//	CAN[myCan].DoubleLoad 	:= FALSE;
//END_IF;

//Bag Ready to Washing Machine
IF (step = 5) THEN
	o_bagReady 			:= myPushButtonControl OR myPickerControl;
	IF (myCan > 0) THEN CAN[myCan].BagReady := NOT myPushButtonControl OR myPickerControl; END_IF;
	IF i_openBag OR TestDischarger THEN
		D[900 + mySeq] := 6;
	END_IF;
ELSE
	CAN[myCan].BagReady	:= FALSE;
END_IF;

//Set LoadDropped to False
IF (step <> 6) THEN
	LoadDropped := FALSE;
END_IF;

//Open Bag Until LoadDropped Received and has been open for 6 seconds
ton_10ms_MinOpen(IN:= (step = 6), PT:= 600);
IF (step = 6) THEN

	IF (myPushButtonControl OR myPickerControl) THEN
		IF (NOT i_openBag OR TestDischarger) THEN
			LoadDropped := TRUE;
		END_IF;
	ELSE
		IF (i_loadDropped OR TestDischarger) THEN
			LoadDropped := TRUE;
		END_IF;
	END_IF;

	IF (LoadDropped AND ton_10ms_MinOpen.Q) THEN
//		//Write Report
//		IF (ReportUnloading[myDC].Cat = 0) THEN
//			ReportUnloading[myDC].Prg := bag.Prg; 	//Program
//			ReportUnloading[myDC].Cat := bag.Cat;	//Category
//			ReportUnloading[myDC].Cus := bag.Cus;	//Customer
//			ReportUnloading[myDC].Wgt := bag.Wgt;	//Weight
//			ReportUnloading[myDC].Cnt := 0;					//Count
//			ReportUnloading[myDC].Stn := 0;					//Station
//			ReportUnloading[myDC].Mcn := myDC;				//Machine
//			ReportUnloading[myDC].Mis := bag.Mis;	//Batch ID
//			D[batchSizeSet] := (D[batchSizeSet] - 1);
//		END_IF
		D[900 + mySeq] := 7;
		alarm.Time := 60000;
		alarm.Name := almLoadNotDropped;
	END_IF;
END_IF;

//Change display to empty bag - clear all other bag data
IF (step = 7) THEN
	IF myPushButtonControl THEN
		o_bagReady := Std.Clock200ms;
		IF ((NOT i_openBag AND NOT i_loadDropped AND NOT i_bagEmpty) OR TestDrop) THEN
			//bag		:= Bag[0];
			bag.Prg 	:= Std.MaxProg;
			bag.Cat	:= Std.MaxCats;
			bag.Cus 	:= Std.MaxCust;
			bag.Dst 	:= 0;
			D[900 + mySeq] 	:= 8;
		END_IF;
		IF (i_loadDropped OR i_bagEmpty) THEN
			alarm.Name := ALM_SWITCH_FAULT;
		END_IF;
	ELSE
		IF ((NOT i_openBag AND NOT i_loadDropped AND NOT i_bagEmpty) OR TestDrop) THEN
			//bag		:= Bag[0];
			bag.Prg 	:= Std.MaxProg;
			bag.Cat	:= Std.MaxCats;
			bag.Cus 	:= Std.MaxCust;
			bag.Dst 	:= 0;
			D[900 + mySeq] 	:= 8;
		END_IF;
		IF (i_openBag OR i_loadDropped OR i_bagEmpty) THEN
			alarm.Name := almSwitchFault;
		END_IF;
	END_IF;
END_IF;

//Close bag
ton_10ms_CloserDelay(IN:= (step = 8), PT:= 200);
ton_10ms_CloserDown(IN:= (step = 8), PT:= 800);
IF (step = 8) THEN
	IF myBagCloser THEN
		o_closer := ton_10ms_CloserDelay.Q;
		IF ton_10ms_CloserDown.Q THEN
			D[900 + mySeq] := 9;
		END_IF;
	ELSE
		D[900 + mySeq] := 10;
	END_IF;
END_IF;

//Allow closer to go back up
ton_10ms_CloserUp(IN:= (step = 9), PT:= 600);
IF (step = 9) THEN
	IF ton_10ms_CloserUp.Q THEN
		D[900 + mySeq] := 10;
	END_IF;
END_IF;

//Allow steadys to go up
ton_10ms_SteadyUp(IN:= (step = 10), PT:= 200);
IF (step = 10) THEN
	IF ton_10ms_SteadyUp.Q AND NOT EnableRel.DC[myDC] THEN
		D[900 + mySeq] := 11;
	END_IF;
END_IF;

//Check for space on empty bag buffer / Request release
UseCounter := (myRelCounter > 0);
IF (step = 11) THEN
	IF UseCounter THEN
		IF (Line[myRelCounter].Clear AND NOT i_bagAtEmptyBuffer AND NOT o_emptyBagBufferOpen) THEN
			D[900 + mySeq] := 12;
		END_IF;
		IF (Line[myRelCounter].Clear AND i_bagAtEmptyBuffer AND NOT o_emptyBagBufferOpen) THEN
			alarm.Name := almSwitchFault;
		END_IF;
	ELSE
		RequestRel.DC[myDC]	:= TRUE;
		IF EnableRel.DC[myDC] THEN
			D[900 + mySeq] := 12;
		END_IF;
	END_IF;
END_IF;

//Open buffer stop - unitl bag out
IF (step = 12) THEN
	o_openStop := (((outBag.Cat = 0) AND (bag.Cat > 0)) OR (myOutBag = 0));
	IF (myOutBag = 0) THEN
		bag := Bag[0]; //Clear bag;
	END_IF;

	IF UseCounter THEN
		IF pls THEN
			C[myRelCounter] := 0;
		END_IF;
		IF (myOutBag > 0) THEN
			IF (outBag.Cat = 0) AND (bag.Cat > 0) AND Line[myRelCounter].Trip  THEN
				outBag := bag;
				bag := Bag[0];
				D[900 + mySeq] := 1;
			END_IF;
		ELSE
			IF Line[myRelCounter].Trip OR i_bagReleased  THEN
				D[900 + mySeq] := 1;
			END_IF;
		END_IF;
	ELSE
		IF NOT EnableRel.DC[myDC] AND ((myOutBag = 0) OR (bag.Cat = 0)) THEN
			D[900 + mySeq] := 1;
		END_IF;
	END_IF;
	alarm.Name := almBagNotReleased;
END_IF;

//Alarms
timerAlarm(IN := NOT pls AND (alarm.Name > 0),PT:= alarm.Time);
alarm.On 	:= timerAlarm.Q;
alarm.ET 	:= timerAlarm.ET;

//Outputs
Request.SK[myDC] := o_bagReady;
Y[myIO].Y01 	:= o_openBuffer;
Y[myIO].Y02 	:= o_steadys;
Y[myIO].Y03 	:= o_openBag;
Y[myIO].Y04 	:= o_openStop;
Y[myIO].Y05 	:= o_closer;
END_PROGRAM
```

### Program Logical/BaseStandards/Discharger/withStaticBag/x_sb (IEC, version 1.00.2) - *Static bag -- Pushbutton controls

#### staticBag.st - Implementation code
```iecst
(********************************************************************
* COPYRIGHT --
********************************************************************
* PROGRAM: sb
* File: sb.st
* Author: treamsbottom
* Created: March 16, 2018
********************************************************************
* Implementation OF Static Bag
********************************************************************)
//V1.00.1 First Release
//V1.00.2 Add option to use Comms or Pushbutton via the myCan Var.
PROGRAM _INIT
//Configuration
mySeq						:= 23;	//Sequence number
myZone						:= 0;

myDC						:= 14;// Discharger Static bag is linked to
myIO						:= 150 + myDC; // use standard numbering or override with manual reference.
myBag						:= 296; //Buffer Bag
myDischargerBag				:= 295;
myCan						:= myDC;  // If use the myCan we enable automatic release from the discharger.

alarm						ACCESS ADR(Alarm[mySeq]);
bag							ACCESS ADR(Bag[myBag]);
bag_disch					ACCESS ADR(Bag[myDischargerBag]);
can							ACCESS ADR(CAN[myCan]);

END_PROGRAM

PROGRAM _CYCLIC
//Inputs
i_pushbutton 	:= X[myIO].X05;
pushbutton.CLK 	:= i_pushbutton;
pushbutton();

staticBagEnable := NOT Std.HaltSysZone[myZone];

o_bagReady 					:= 0;
o_openBag 					:= 0;
o_openCatch 				:= 0;
Enable.SK[myDC]				:= 0;
IF (myCan > 0) THEN
	can.BagReady 			:= 0;
END_IF;

IF (myBag = 0) THEN
	alarm.Bag	:= mySeq + 10000;
ELSE
	alarm.Bag	:= myBag;
END_IF;

alarm.Name 		:= 0;
alarm.Beacon	:= TRUE;
alarm.Extra		:= 0;
alarm.Time		:= 3000;

//Setup Sequence
step := D[900 + mySeq];
//Setup Pulse contact
pls := (step <> laststep);
laststep := step;

//Sequence
IF (step = 0) THEN
	//Disabled
END_IF;

//step 1 - Check signals
IF (step = 1) THEN
	IF staticBagEnable THEN
		IF (myCan > 0) THEN
			IF NOT can.DropLoad AND NOT can.LoadDropped THEN
				D[900 + mySeq] := 2;
			ELSE
				alarm.Name := ALM_SWITCH_FAULT;
				alarm.Time := 0;
			END_IF;
		ELSIF (NOT i_pushbutton AND (bag.Cat = 0)) THEN
			D[900 + mySeq] := 2;
		END_IF;
		IF (bag.Cat <> 0) THEN
			alarm.Name := ALM_BAG_DATA_ERROR;
			alarm.Time := 0;
		ELSIF i_pushbutton AND (myCan = 0) THEN
			alarm.Name := ALM_SWITCH_FAULT;
			alarm.Time := 0;
		END_IF;
	END_IF;
END_IF;

IF (bag.Cat > 0) AND (bag.Bid = 0) AND (BidStn > 0) THEN
	bag.Bid := BidStn;
	BidStn := 0;
END_IF;

//step 2 - Enable discharger TO open
IF (step = 2) THEN
	IF (myCan > 0) THEN // Release from Discharger automatically
		IF (Request.SK[myDC] AND (bag_disch.Cat > 0) AND (bag.Cat = 0)) THEN
			bag := bag_disch;
			bag_disch.Cat :=  Std.MaxCats;
			bag_disch.Prg 	:= Std.MaxProg;
			bag_disch.Cus	:= Std.MaxCust;
			bag_disch.Dst := 0;
			bag.Bid := 0;
			D[900 + mySeq] := 3;
		ELSIF Request.SK[myDC] AND (bag_disch.Cat = 0) THEN
			alarm.Name := ALM_BAG_DATA_ERROR;
			alarm.Time := 0;
			alarm.Bag := myDischargerBag;
		ELSIF (bag.Cat > 0) THEN
			alarm.Name := ALM_BAG_DATA_ERROR;
			alarm.Time := 0;
		END_IF;
	ELSE //Pushbutton
		o_bagReady := Request.SK[myDC] AND Std.Clock2s AND (bag_disch.Cat > 0);
		IF (Request.SK[myDC] AND pushbutton.Q AND (bag_disch.Cat > 0)) THEN
			bag := bag_disch;
			bag_disch.Cat :=  Std.MaxCats;
			bag_disch.Prg 	:= Std.MaxProg;
			bag_disch.Cus	:= Std.MaxCust;
			bag_disch.Dst := 0;
			bag.Bid := 0;
			D[900 + mySeq] := 3;
		ELSIF Request.SK[myDC] AND (bag_disch.Cat = 0) THEN
			alarm.Name := ALM_BAG_DATA_ERROR;
			alarm.Time := 0;
			alarm.Bag := myDischargerBag;
		END_IF;
	END_IF;

END_IF;

//step 3 - Allow linen TO drop
ton_10ms_MinDischOpen(IN:= NOT Request.SK[myDC],PT:= 100);
IF (step = 3) THEN
	o_openCatch 	:= 1;
	Enable.SK[myDC] := 1;
	IF ton_10ms_MinDischOpen.Q THEN
		D[900 + mySeq] := 4;
	END_IF;
END_IF;

codeStep  := ((step >= 4) AND (step <= 5));

//Wash Codes
IF codeStep THEN
	can.Program		:= bag.Prg;
	can.Category 	:= bag.Cat;
	can.Customer 	:= bag.Cus;
	can.Weight   	:= bag.Wgt;
	can.BatchID		:= bag.Mis;
	can.DoubleLoad 	:= FALSE;
ELSE
	can.Program 	:= 0;
	can.Category 	:= 0;
	can.Customer 	:= 0;
	can.Weight   	:= 0;
	can.BatchID		:= 0;
	can.DoubleLoad 	:= FALSE;
END_IF;

//step 4 - Bag full wait Drop load from Washing Machine
IF (step = 4) THEN
	o_bagReady := (myCan = 0);
	can.BagReady := (myCan > 0);
	IF (myCan > 0) THEN
		IF can.DropLoad THEN
			D[900 + mySeq] := 5;
		END_IF;
	ELSIF pushbutton.Q THEN
		D[900 + mySeq] := 5;
	END_IF;
END_IF;

//step 5 - Open bag
ton_10ms_minOpen(IN:= (step = 5),PT:= 600);
IF (step = 5) THEN
	o_openCatch 	:= TRUE;
	o_openBag 		:= TRUE;
	IF (myCan > 0) THEN
		IF can.LoadDropped THEN
			loadDropped := 1;
		END_IF;
	ELSE
		o_bagReady 		:= Std.Clock1s AND ton_10ms_minOpen.Q;
		IF  pushbutton.Q  AND ton_10ms_minOpen.Q THEN
			loadDropped := 1;
		END_IF;
	END_IF;

	IF loadDropped AND ton_10ms_minOpen.Q THEN
		//Write Report
		IF (ReportUnloading[myDC].Cat = 0) AND Std.StationReports THEN
			ReportUnloading[myDC].Prg := bag.Prg;// 	;PROGRAM
			ReportUnloading[myDC].Cus := bag.Cus;//		;Customer
			ReportUnloading[myDC].Wgt := bag.Wgt;//		;Weight
			ReportUnloading[myDC].Cnt := 0;//			;Count
			ReportUnloading[myDC].Stn := 0;//			;Station
			ReportUnloading[myDC].Mcn := myDC;//		;Machine
			ReportUnloading[myDC].Bid := bag.Bid;//
			ReportUnloading[myDC].Mis := bag.Mis;//		;Batch ID
			//ReportUnloading[myDC].TimeStamp := CurrentTimestamp;//
			bag := Bag[0];
			D[900 + mySeq] := 6;
		END_IF;
	END_IF;
ELSE
	loadDropped := 0;
END_IF;

//step 6 - Close bag
ton_10ms_closerDown(IN:= (step = 6),PT:= 1000);
IF (step = 6) THEN
	o_openCatch := TRUE;
	IF ton_10ms_closerDown.Q THEN
		bag := Bag[0];
		D[900 + mySeq] := 7;
	END_IF;
END_IF;

//step 7 - Allow catch TO settle
ton_10ms_closerUp(IN:= (step = 7),PT:= 400);
IF (step = 7) THEN
	IF ton_10ms_closerUp.Q THEN
		D[900 + mySeq] := 1;
	END_IF;
END_IF;

//-----------------------------------
//PLC Outputs - adjust TO suit system
//-----------------------------------

Y[myIO].Y08	:= o_bagReady  AND (myCan = 0);
Y[myIO].Y06	:= o_openCatch;
Y[myIO].Y07 := o_openBag;

//Alarms
timerAlarm(IN := NOT pls AND (alarm.Name > 0),PT:= alarm.Time);

alarm.On 	:= timerAlarm.Q;
alarm.ET 	:= timerAlarm.ET;

END_PROGRAM
```

#### staticBag.var - Local variables
```iecst
(********************************************************************
 * COPYRIGHT --
 ********************************************************************
 * Program: pr
 * File: pr.var
 * Author: treamsbottom
 * Created: July 16, 2015
 ********************************************************************
 * Local variables of program pr
 ********************************************************************)
VAR
	mySeq : UINT;
	myZone : UINT;
	myBag : UINT;
	step : UINT;
	pls : BOOL;
	timerAlarm : TON_10ms;
END_VAR
VAR RETAIN
	lastStep : UINT;
END_VAR
VAR
	alarm : REFERENCE TO Alm;
	bag : REFERENCE TO Bag_typ;
	myDC : UINT;
	myIO : UINT;
	myDischargerBag : UINT;
	bag_disch : REFERENCE TO Bag_typ;
	i_pushbutton : BOOL;
	o_bagReady : BOOL;
	o_openCatch : BOOL;
	o_openBag : BOOL;
	pushbutton : F_TRIG;
	staticBagEnable : BOOL;
	ton_10ms_MinDischOpen : TON_10ms;
	laststep : UINT;
	loadDropped : BOOL;
	ton_10ms_minOpen : TON_10ms;
	ton_10ms_closerDown : TON_10ms;
	ton_10ms_closerUp : TON_10ms;
	myCan : UINT;
	can : REFERENCE TO CAN_Vars;
	codeStep : BOOL;
END_VAR
```

### Package Logical/BaseStandards/Empty - *Empty Base Sequence

### Program Logical/BaseStandards/Empty/empty (IEC, version 1.00.1) - *Empty base sequence

#### empty.st - Implementation code
```iecst
(********************************************************************
 * COPYRIGHT --
 ********************************************************************
 * Program: pr
 * File: pr.st
 * Author: treamsbottom
 * Created: July 16, 2015
 ********************************************************************
 * Implementation of program pr
 ********************************************************************)
//V1.00.1 First Release
PROGRAM _INIT
//Configuration
mySeq						:= 22;	//Sequence number
myIO						:= 220;
myZone						:= 0;
myRelLine					:= 22;
myBag						:= 255; //Buffer Bag
//myBuffBag					:= 0;
//myOutBag 					:= Line[myRelLine].LastBag;
//myCan						:= 0;
bufferSettleTime			:= 300;

alarm						ACCESS ADR(Alarm[mySeq]);
bag							ACCESS ADR(Bag[myBag]);
//bag_buff					ACCESS ADR(Bag[myBuffBag]);
//bag_out						ACCESS ADR(Bag[myOutBag]);
//can							ACCESS ADR(CAN[myCan]);
line_release				ACCESS ADR(Line[myRelLine]);

END_PROGRAM

PROGRAM _CYCLIC
//Inputs
i_bagAtBuffer				:= X[myIO].X01;

i_bagAtBufferOut 		:= FALSE; // Any Single bag buffer out IO.
i_bufferOutOpen			:= FALSE;

o_openBuffer			:= FALSE;

IF (myBag = 0) THEN
	alarm.Bag	:= mySeq + 10000;
ELSE
	alarm.Bag	:= myBag;
END_IF;

alarm.Name 		:= 0;
alarm.Beacon	:= TRUE;
alarm.Extra		:= 0;
alarm.Time		:= 3000;

//Setup Sequence
step := D[900 + mySeq];
//Setup Pulse contact
pls := (step <> lastStep);
lastStep := step;

//Sequence
IF (step = 0) THEN
	//Disabled
END_IF;

//-----------------------------------
//PLC Outputs - adjust TO suit system
//-----------------------------------

Y[myIO].Y05 := o_openBuffer;

//Alarms
timerAlarm(IN := NOT pls AND (alarm.Name > 0),PT:= alarm.Time);

alarm.On 	:= timerAlarm.Q;
alarm.ET 	:= timerAlarm.ET;

END_PROGRAM
```
